--- Backups/Rob4/HOME/Module1.mod ---
MODULE Module1
!PERS tooldata DrillTool:=[TRUE,[[31.792631019,0,229.638935148],[0.945518576,0,0.325568154,0]],[1,[0,0,1],[1,0,0,0],0,0,0]];
PERS tooldata DrillTool:=[TRUE,[[67.056,0,55.372],[0.7071,0,0.7071,0]],[1,[0,0,1],[1,0,0,0],0,0,0]];
PERS wobjdata FakeWing:=[FALSE, TRUE, "",[[-738.2, -596.9, 290],[0.9912, 0, -0.1326, 0]],[[0, 0, 0],[1, 0, 0, 0]]];
!PERS wobjdata FakeWing:=[FALSE, TRUE, "",[[-738.2, -871.22, 290],[1,0,0,0]],[[0, 0, 0],[1, 0, 0, 0]]];
CONST jointtarget jHome:=[[-90,0,28.434410486,3.185484116,-20,-3.571881577],[9E+09,9E+09,9E+09,9E+09,9E+09,9E+09]];
	CONST robtarget Target_10:=[[968.8,4.8,-256.8],[-0.107942386345314,0.559135464335052,0.818413471745805,-0.0769113971910747],[-1,0,0,1],[9E+09,9E+09,9E+09,9E+09,9E+09,9E+09]];
	CONST robtarget Target_20:=[[968.8,9.6,-256.9],[-0.106640376548865,0.55772059756557,0.819364658230691,-0.0788487284813297],[-1,0,0,1],[9E+09,9E+09,9E+09,9E+09,9E+09,9E+09]];
	CONST robtarget Target_30:=[[968.8,14.5,-256.9],[-0.105307817924908,0.556255492926737,0.820340422972373,-0.0808188128484617],[-1,0,0,1],[9E+09,9E+09,9E+09,9E+09,9E+09,9E+09]];
	CONST robtarget Target_40:=[[968.8,19.3,-257],[-0.104018956602322,0.554797112975153,0.821298505042471,-0.0827585990504985],[-1,0,0,1],[9E+09,9E+09,9E+09,9E+09,9E+09,9E+09]];
	CONST robtarget Target_50:=[[968.8,24.1,-257.1],[-0.10270808792262,0.553310583836471,0.822263480299647,-0.0847420524611851],[-1,0,0,1],[9E+09,9E+09,9E+09,9E+09,9E+09,9E+09]];
	CONST robtarget Target_60:=[[968.8,28.9,-257.3],[-0.101414305361901,0.551800115908394,0.823230694611851,-0.0867351958569063],[-1,0,0,1],[9E+09,9E+09,9E+09,9E+09,9E+09,9E+09]];
	CONST robtarget Target_70:=[[968.8,33.7,-257.4],[-0.100146565654331,0.55027415284443,0.824199705211674,-0.0886784530084809],[-1,0,0,1],[9E+09,9E+09,9E+09,9E+09,9E+09,9E+09]];
	CONST robtarget Target_80:=[[968.8,38.5,-257.6],[-0.0988674093110697,0.54871723908215,0.825174424011152,-0.0906741245783206],[-1,0,0,1],[9E+09,9E+09,9E+09,9E+09,9E+09,9E+09]];
	CONST robtarget Target_90:=[[968.8,43.4,-257.8],[-0.0976274781322347,0.547116328064163,0.826167750273506,-0.0926253069476237],[-1,0,0,1],[9E+09,9E+09,9E+09,9E+09,9E+09,9E+09]];
	CONST robtarget Target_100:=[[968.8,48.2,-258.1],[-0.0963734022079838,0.545509328348709,0.827149560398508,-0.0946326833813457],[-1,0,0,1],[9E+09,9E+09,9E+09,9E+09,9E+09,9E+09]];
	CONST robtarget Target_110:=[[968.8,53,-258.3],[-0.0951272887762192,0.543877494214756,0.828135551386225,-0.0966414959890247],[-1,0,0,1],[9E+09,9E+09,9E+09,9E+09,9E+09,9E+09]];
	CONST robtarget Target_120:=[[968.8,57.8,-258.6],[-0.0939178195285495,0.54222699826944,0.82912338791337,-0.0986089911609059],[-1,0,0,1],[9E+09,9E+09,9E+09,9E+09,9E+09,9E+09]];
	CONST robtarget Target_130:=[[968.8,62.6,-258.9],[-0.0926884156537042,0.540544275757953,0.83011823749075,-0.100620352484805],[-1,0,0,1],[9E+09,9E+09,9E+09,9E+09,9E+09,9E+09]];
	CONST robtarget Target_140:=[[968.8,67.4,-259.2],[-0.091496096140411,0.538842149319605,0.831115432114365,-0.102590160390974],[-1,0,0,1],[9E+09,9E+09,9E+09,9E+09,9E+09,9E+09]];
	CONST robtarget Target_150:=[[968.8,72.3,-259.6],[-0.0902970417660465,0.537075607015845,0.832137487086423,-0.104610894185818],[-1,0,0,1],[9E+09,9E+09,9E+09,9E+09,9E+09,9E+09]];
	CONST robtarget Target_160:=[[968.8,77.1,-260],[-0.0891036215361824,0.535310554276655,0.833145780021638,-0.106636130562277],[-1,0,0,1],[9E+09,9E+09,9E+09,9E+09,9E+09,9E+09]];
	CONST robtarget Target_170:=[[968.8,81.9,-260.4],[-0.0879477385246057,0.533524737247738,0.834157223840012,-0.108619869032618],[-1,0,0,1],[9E+09,9E+09,9E+09,9E+09,9E+09,9E+09]];
	CONST robtarget Target_180:=[[968.8,86.7,-260.8],[-0.0867820002749409,0.531701655816364,0.835174793612655,-0.110658473441827],[-1,0,0,1],[9E+09,9E+09,9E+09,9E+09,9E+09,9E+09]];
	CONST robtarget Target_190:=[[968.8,91.5,-261.3],[-0.0856457062027853,0.529858976157848,0.836197037860416,-0.11264453944799],[-1,0,0,1],[9E+09,9E+09,9E+09,9E+09,9E+09,9E+09]];
	CONST robtarget Target_200:=[[968.8,96.3,-261.8],[-0.0845001294653035,0.52797768348931,0.837225467326941,-0.114685704064607],[-1,0,0,1],[9E+09,9E+09,9E+09,9E+09,9E+09,9E+09]];
	CONST robtarget Target_210:=[[968.8,101.2,-262.3],[-0.0833777397174588,0.526031720385176,0.83827881205061,-0.11673651928697],[-1,0,0,1],[9E+09,9E+09,9E+09,9E+09,9E+09,9E+09]];
	CONST robtarget Target_220:=[[968.8,106,-262.8],[-0.0822813203856298,0.524096558354244,0.839317580280092,-0.118737446787462],[-1,0,0,1],[9E+09,9E+09,9E+09,9E+09,9E+09,9E+09]];
	CONST robtarget Target_230:=[[968.8,110.8,-263.4],[-0.0811763419641853,0.522120475519326,0.840362638876055,-0.12079422887729],[-1,0,0,1],[9E+09,9E+09,9E+09,9E+09,9E+09,9E+09]];
	CONST robtarget Target_240:=[[968.8,115.6,-264],[-0.0801102368360122,0.520119946233772,0.841412748073788,-0.122809522687666],[-1,0,0,1],[9E+09,9E+09,9E+09,9E+09,9E+09,9E+09]];
	CONST robtarget Target_250:=[[968.8,120.4,-264.6],[-0.0790283539545263,0.518079466998265,0.842470151681068,-0.124868845884432],[-1,0,0,1],[9E+09,9E+09,9E+09,9E+09,9E+09,9E+09]];
	CONST robtarget Target_260:=[[968.8,125.3,-265.2],[-0.0779715226802002,0.515967795467923,0.843554530052155,-0.126938688032417],[-1,0,0,1],[9E+09,9E+09,9E+09,9E+09,9E+09,9E+09]];
	CONST robtarget Target_270:=[[968.8,130.1,-265.9],[-0.076949075572964,0.513864462728356,0.844623466676326,-0.128970358040245],[-1,0,0,1],[9E+09,9E+09,9E+09,9E+09,9E+09,9E+09]];
	CONST robtarget Target_280:=[[968.8,134.9,-266.6],[-0.0759120858706762,0.511718820666067,0.845699772579321,-0.131046169170174],[-1,0,0,1],[9E+09,9E+09,9E+09,9E+09,9E+09,9E+09]];
	CONST robtarget Target_290:=[[968.8,139.7,-267.3],[-0.0748882393420013,0.509537785767557,0.846782863288632,-0.133123172002685],[-1,0,0,1],[9E+09,9E+09,9E+09,9E+09,9E+09,9E+09]];
	CONST robtarget Target_300:=[[968.8,144.5,-268],[-0.0739120235779645,0.507325477212431,0.847871706099419,-0.135171901436095],[-1,0,0,1],[9E+09,9E+09,9E+09,9E+09,9E+09,9E+09]];
	CONST robtarget Target_310:=[[968.8,149.4,-268.8],[-0.0729217598159667,0.505032843902239,0.848991917508329,-0.137247832518004],[-1,0,0,1],[9E+09,9E+09,9E+09,9E+09,9E+09,9E+09]];
	CONST robtarget Target_320:=[[968.8,154.2,-269.6],[-0.0719805492460282,0.502742088257011,0.850094765604421,-0.139312895014009],[-1,0,0,1],[9E+09,9E+09,9E+09,9E+09,9E+09,9E+09]];
	CONST robtarget Target_330:=[[968.8,159,-270.4],[-0.0710201466278696,0.500407925392313,0.851206058488137,-0.141408249301824],[-1,0,0,1],[9E+09,9E+09,9E+09,9E+09,9E+09,9E+09]];
	CONST robtarget Target_340:=[[968.8,163.8,-271.2],[-0.0701081554829596,0.498039124477821,0.852324167132108,-0.143476099566102],[-1,0,0,1],[9E+09,9E+09,9E+09,9E+09,9E+09,9E+09]];
	CONST robtarget Target_350:=[[968.8,168.6,-272.1],[-0.0691850402824734,0.495621840436952,0.853449773615657,-0.145588136186932],[-1,0,0,1],[9E+09,9E+09,9E+09,9E+09,9E+09,9E+09]];
	CONST robtarget Target_360:=[[968.8,173.4,-273],[-0.0682778424968577,0.493163293359647,0.854583178611091,-0.147701364724926],[-1,0,0,1],[9E+09,9E+09,9E+09,9E+09,9E+09,9E+09]];
	CONST robtarget Target_370:=[[968.8,178.3,-273.9],[-0.0674207080420315,0.490627737512659,0.855749964564331,-0.149769387587943],[-1,0,0,1],[9E+09,9E+09,9E+09,9E+09,9E+09,9E+09]];
	CONST robtarget Target_380:=[[968.8,183.1,-274.9],[-0.0665534629922089,0.488079478410023,0.85689877770681,-0.151899783025914],[-1,0,0,1],[9E+09,9E+09,9E+09,9E+09,9E+09,9E+09]];
	CONST robtarget Target_390:=[[968.8,187.9,-275.8],[-0.0657293478681176,0.485495470345176,0.85805671857293,-0.153988534686852],[-1,0,0,1],[9E+09,9E+09,9E+09,9E+09,9E+09,9E+09]];
	CONST robtarget Target_400:=[[968.8,192.7,-276.8],[-0.0648970915608762,0.482857906815298,0.859222188208384,-0.156121236938751],[-1,0,0,1],[9E+09,9E+09,9E+09,9E+09,9E+09,9E+09]];
	CONST robtarget Target_410:=[[968.8,197.5,-277.9],[-0.0640894833612442,0.480170166912685,0.860394987305689,-0.158270700853872],[-1,0,0,1],[9E+09,9E+09,9E+09,9E+09,9E+09,9E+09]];
	CONST robtarget Target_420:=[[973.5,197.2,-279.1],[-0.0647831891782489,0.476538276592348,0.862417809926292,-0.157955469877521],[-1,0,0,1],[9E+09,9E+09,9E+09,9E+09,9E+09,9E+09]];
	CONST robtarget Target_430:=[[978.2,197,-280.4],[-0.0654513013274054,0.472883025030647,0.864427470973437,-0.157679799653864],[-1,0,0,1],[9E+09,9E+09,9E+09,9E+09,9E+09,9E+09]];
	CONST robtarget Target_440:=[[982.9,196.6,-281.6],[-0.0660933755521842,0.46935615793945,0.866347508185939,-0.157411745979934],[-1,0,0,1],[9E+09,9E+09,9E+09,9E+09,9E+09,9E+09]];
	CONST robtarget Target_450:=[[987.6,196.4,-282.9],[-0.0667443729406992,0.465766124616528,0.86828286007232,-0.157136821735347],[-1,0,0,1],[9E+09,9E+09,9E+09,9E+09,9E+09,9E+09]];
	CONST robtarget Target_460:=[[992.3,196.1,-284.1],[-0.0674028023794809,0.462266046873075,0.870157221438666,-0.156822747450342],[-1,0,0,1],[9E+09,9E+09,9E+09,9E+09,9E+09,9E+09]];
	CONST robtarget Target_470:=[[997.1,195.8,-285.4],[-0.0680417113457267,0.458714001293542,0.87203494948929,-0.156546598186054],[-1,0,0,1],[9E+09,9E+09,9E+09,9E+09,9E+09,9E+09]];
	CONST robtarget Target_480:=[[1001.8,195.5,-286.6],[-0.0686583135132066,0.455272740455241,0.873836494953086,-0.156277150831474],[-1,0,0,1],[9E+09,9E+09,9E+09,9E+09,9E+09,9E+09]];
	CONST robtarget Target_490:=[[1006.5,195.2,-287.9],[-0.0692598520335908,0.451868831293863,0.875604850746204,-0.155992876603775],[-1,0,0,1],[9E+09,9E+09,9E+09,9E+09,9E+09,9E+09]];
	CONST robtarget Target_500:=[[1011.2,194.9,-289.1],[-0.0698599262628231,0.448494319419836,0.877338099476652,-0.155725063356508],[-1,0,0,1],[9E+09,9E+09,9E+09,9E+09,9E+09,9E+09]];
	CONST robtarget Target_510:=[[1015.9,194.6,-290.4],[-0.0704757269732864,0.445161665334504,0.879039624191811,-0.155414293824337],[-1,0,0,1],[9E+09,9E+09,9E+09,9E+09,9E+09,9E+09]];
	CONST robtarget Target_520:=[[1020.6,194.3,-291.6],[-0.0710595030740004,0.441853803362528,0.880706980576819,-0.155148244721643],[-1,0,0,1],[9E+09,9E+09,9E+09,9E+09,9E+09,9E+09]];
	CONST robtarget Target_530:=[[1025.3,194,-292.9],[-0.0716353435846854,0.438579183432016,0.882342262981194,-0.154883208795643],[-1,0,0,1],[9E+09,9E+09,9E+09,9E+09,9E+09,9E+09]];
	CONST robtarget Target_540:=[[1030.1,193.7,-294.1],[-0.0722159183465569,0.435265792974258,0.883981480942423,-0.154613362794727],[-1,0,0,1],[9E+09,9E+09,9E+09,9E+09,9E+09,9E+09]];
	CONST robtarget Target_550:=[[1034.8,193.4,-295.4],[-0.0727991731829624,0.432066562567872,0.885555376103445,-0.15430632439711],[-1,0,0,1],[9E+09,9E+09,9E+09,9E+09,9E+09,9E+09]];
	CONST robtarget Target_560:=[[1039.5,193.1,-296.6],[-0.0733514213142073,0.428891789433335,0.887097329266413,-0.154044572628362],[-1,0,0,1],[9E+09,9E+09,9E+09,9E+09,9E+09,9E+09]];
	CONST robtarget Target_570:=[[1044.2,192.8,-297.9],[-0.0738960968592212,0.425749832850519,0.888609542185254,-0.153784031141213],[-1,0,0,1],[9E+09,9E+09,9E+09,9E+09,9E+09,9E+09]];
	CONST robtarget Target_580:=[[1048.9,192.5,-299.1],[-0.0744560047898698,0.422649013071223,0.890094329524097,-0.153480290753246],[-1,0,0,1],[9E+09,9E+09,9E+09,9E+09,9E+09,9E+09]];
	CONST robtarget Target_590:=[[1053.6,192.3,-300.4],[-0.0749948386695809,0.41951882253895,0.89157392359611,-0.153217722447156],[-1,0,0,1],[9E+09,9E+09,9E+09,9E+09,9E+09,9E+09]];
	CONST robtarget Target_600:=[[1058.4,191.9,-301.6],[-0.0755196426375664,0.416459958972194,0.893006834393729,-0.152959732854318],[-1,0,0,1],[9E+09,9E+09,9E+09,9E+09,9E+09,9E+09]];
	CONST robtarget Target_610:=[[1063.2,191.7,-302.9],[-0.0760553161680778,0.413327332533263,0.894461077902201,-0.152694090198487],[-1,0,0,1],[9E+09,9E+09,9E+09,9E+09,9E+09,9E+09]];
	CONST robtarget Target_620:=[[1063.2,186.7,-301.8],[-0.0766806108289428,0.416479421442643,0.893328220646938,-0.150431597855895],[-1,0,0,1],[9E+09,9E+09,9E+09,9E+09,9E+09,9E+09]];
	CONST robtarget Target_630:=[[1063.2,181.8,-300.8],[-0.0773349992657743,0.419532651685502,0.892221234188017,-0.148165182557526],[-1,0,0,1],[9E+09,9E+09,9E+09,9E+09,9E+09,9E+09]];
	CONST robtarget Target_640:=[[1063.2,176.9,-299.8],[-0.078016434697904,0.422537939615321,0.891114002676915,-0.145914220471464],[-1,0,0,1],[9E+09,9E+09,9E+09,9E+09,9E+09,9E+09]];
	CONST robtarget Target_650:=[[1063.2,172,-298.9],[-0.0787092090169855,0.425503303914037,0.890009339895156,-0.143649481981481],[-1,0,0,1],[9E+09,9E+09,9E+09,9E+09,9E+09,9E+09]];
	CONST robtarget Target_660:=[[1063.2,167.1,-298],[-0.0794359651980819,0.428418799418737,0.888903404145049,-0.141414277344971],[-1,0,0,1],[9E+09,9E+09,9E+09,9E+09,9E+09,9E+09]];
	CONST robtarget Target_670:=[[1063.2,162.2,-297],[-0.080173119410487,0.431295682248896,0.887800214850835,-0.139165670724727],[-1,0,0,1],[9E+09,9E+09,9E+09,9E+09,9E+09,9E+09]];
	CONST robtarget Target_680:=[[1063.2,157.3,-296.2],[-0.0809358269586631,0.434127793589296,0.886697299437008,-0.136931917093582],[-1,0,0,1],[9E+09,9E+09,9E+09,9E+09,9E+09,9E+09]];
	CONST robtarget Target_690:=[[1063.2,152.3,-295.3],[-0.0817086501801631,0.436966661334309,0.885572594947853,-0.134703424030007],[-1,0,0,1],[9E+09,9E+09,9E+09,9E+09,9E+09,9E+09]];
	CONST robtarget Target_700:=[[1063.2,147.4,-294.5],[-0.08250580415254,0.439717260260226,0.884473177381368,-0.13247158866448],[-1,0,0,1],[9E+09,9E+09,9E+09,9E+09,9E+09,9E+09]];
	CONST robtarget Target_710:=[[1063.2,142.5,-293.7],[-0.0833275449806797,0.442425399854024,0.883374314134519,-0.130254009300549],[-1,0,0,1],[9E+09,9E+09,9E+09,9E+09,9E+09,9E+09]];
	CONST robtarget Target_720:=[[1063.2,137.6,-293],[-0.084165466257925,0.445094852551447,0.882277267153493,-0.128037378862409],[-1,0,0,1],[9E+09,9E+09,9E+09,9E+09,9E+09,9E+09]];
	CONST robtarget Target_730:=[[1063.2,132.7,-292.2],[-0.0850191501533236,0.447726204834992,0.881182074536164,-0.125821862676577],[-1,0,0,1],[9E+09,9E+09,9E+09,9E+09,9E+09,9E+09]];
	CONST robtarget Target_740:=[[1063.2,127.8,-291.5],[-0.0859121433611262,0.45032775504269,0.88008875807987,-0.123562917425661],[-1,0,0,1],[9E+09,9E+09,9E+09,9E+09,9E+09,9E+09]];
	CONST robtarget Target_750:=[[1063.2,122.9,-290.8],[-0.086780631442478,0.452874240084196,0.878996243451927,-0.121406954792581],[-1,0,0,1],[9E+09,9E+09,9E+09,9E+09,9E+09,9E+09]];
	CONST robtarget Target_760:=[[1063.2,117.9,-290.2],[-0.0877062031981979,0.455442391239945,0.877883293636171,-0.119166996004373],[-1,0,0,1],[9E+09,9E+09,9E+09,9E+09,9E+09,9E+09]];
	CONST robtarget Target_770:=[[1063.2,113,-289.5],[-0.0886123421515343,0.45791392918028,0.876794047722577,-0.117025143278514],[-1,0,0,1],[9E+09,9E+09,9E+09,9E+09,9E+09,9E+09]];
	CONST robtarget Target_780:=[[1063.2,108.1,-288.9],[-0.0895724613928606,0.460367973564089,0.875707061369707,-0.11478347330409],[-1,0,0,1],[9E+09,9E+09,9E+09,9E+09,9E+09,9E+09]];
	CONST robtarget Target_790:=[[1063.2,103.2,-288.4],[-0.0905306758260853,0.462777522277536,0.874621375658715,-0.112599337697844],[-1,0,0,1],[9E+09,9E+09,9E+09,9E+09,9E+09,9E+09]];
	CONST robtarget Target_800:=[[1063.2,98.3,-287.8],[-0.0914776539191496,0.465145784372994,0.873538533379098,-0.110461164285803],[-1,0,0,1],[9E+09,9E+09,9E+09,9E+09,9E+09,9E+09]];
	CONST robtarget Target_810:=[[1063.2,93.4,-287.3],[-0.0924959019244163,0.467493099310707,0.87245488356131,-0.10824595315336],[-1,0,0,1],[9E+09,9E+09,9E+09,9E+09,9E+09,9E+09]];
	CONST robtarget Target_820:=[[1063.2,88.5,-286.8],[-0.0934775740677943,0.469793072491761,0.871375182242977,-0.106121175814107],[-1,0,0,1],[9E+09,9E+09,9E+09,9E+09,9E+09,9E+09]];
	CONST robtarget Target_830:=[[1063.2,83.5,-286.3],[-0.0945168078179997,0.472113460240636,0.870274451230033,-0.103912623081962],[-1,0,0,1],[9E+09,9E+09,9E+09,9E+09,9E+09,9E+09]];
	CONST robtarget Target_840:=[[1063.2,78.6,-285.9],[-0.0955481155796674,0.47435593029813,0.869197771779048,-0.101745970605763],[-1,0,0,1],[9E+09,9E+09,9E+09,9E+09,9E+09,9E+09]];
	CONST robtarget Target_850:=[[1063.2,73.7,-285.5],[-0.0966006758146477,0.476565156559149,0.868121897640117,-0.0995908219849055],[-1,0,0,1],[9E+09,9E+09,9E+09,9E+09,9E+09,9E+09]];
	CONST robtarget Target_860:=[[1063.2,68.8,-285.1],[-0.0976649286535562,0.47874362573452,0.867047946051864,-0.09743696309361],[-1,0,0,1],[9E+09,9E+09,9E+09,9E+09,9E+09,9E+09]];
	CONST robtarget Target_870:=[[1063.2,63.9,-284.7],[-0.0987405471140935,0.480891783652933,0.865975897316991,-0.0952845319909914],[-1,0,0,1],[9E+09,9E+09,9E+09,9E+09,9E+09,9E+09]];
	CONST robtarget Target_880:=[[1063.2,59,-284.4],[-0.0998272086701067,0.483010067703361,0.864905730830889,-0.0931336656758201],[-1,0,0,1],[9E+09,9E+09,9E+09,9E+09,9E+09,9E+09]];
	CONST robtarget Target_890:=[[1063.2,54.1,-284.1],[-0.100934466374847,0.485097309065803,0.863836217768386,-0.09099353332161],[-1,0,0,1],[9E+09,9E+09,9E+09,9E+09,9E+09,9E+09]];
	CONST robtarget Target_900:=[[1063.2,49.1,-283.8],[-0.102048799399347,0.487190226356418,0.862748992686117,-0.0888588853352571],[-1,0,0,1],[9E+09,9E+09,9E+09,9E+09,9E+09,9E+09]];
	CONST robtarget Target_910:=[[1063.2,44.2,-283.6],[-0.103177151310856,0.4892196127847,0.861683235190265,-0.0867216703379402],[-1,0,0,1],[9E+09,9E+09,9E+09,9E+09,9E+09,9E+09]];
	CONST robtarget Target_920:=[[1063.2,39.3,-283.4],[-0.10432573974925,0.491219543140388,0.860617959114868,-0.0845944969349602],[-1,0,0,1],[9E+09,9E+09,9E+09,9E+09,9E+09,9E+09]];
	CONST robtarget Target_930:=[[1063.2,34.4,-283.2],[-0.105484285502105,0.493191938801291,0.85955435750845,-0.0824686819451414],[-1,0,0,1],[9E+09,9E+09,9E+09,9E+09,9E+09,9E+09]];
	CONST robtarget Target_940:=[[1063.2,29.5,-283],[-0.106652496713291,0.495137184746014,0.858492398121187,-0.0803443563341304],[-1,0,0,1],[9E+09,9E+09,9E+09,9E+09,9E+09,9E+09]];
	CONST robtarget Target_950:=[[1063.2,24.6,-282.8],[-0.107840656413329,0.497054461120178,0.857430708523191,-0.0782293780257217],[-1,0,0,1],[9E+09,9E+09,9E+09,9E+09,9E+09,9E+09]];
	CONST robtarget Target_960:=[[1063.2,19.7,-282.7],[-0.109027458012561,0.498946597101844,0.8563719098455,-0.0761082036798955],[-1,0,0,1],[9E+09,9E+09,9E+09,9E+09,9E+09,9E+09]];
	CONST robtarget Target_970:=[[1063.2,14.7,-282.6],[-0.110231181610952,0.500842889389237,0.855294950614735,-0.0740002310930915],[-1,0,0,1],[9E+09,9E+09,9E+09,9E+09,9E+09,9E+09]];
	CONST robtarget Target_980:=[[1063.2,9.8,-282.6],[-0.111457441458863,0.502680910869204,0.854236489571451,-0.0718968738944611],[-1,0,0,1],[9E+09,9E+09,9E+09,9E+09,9E+09,9E+09]];
	CONST robtarget Target_990:=[[1063.2,4.9,-282.5],[-0.112681393063629,0.504494799312451,0.853180840830537,-0.0697879213304613],[-1,0,0,1],[9E+09,9E+09,9E+09,9E+09,9E+09,9E+09]];
	CONST robtarget Target_1000:=[[1067.8,0,-283.8],[-0.11412479964084,0.503756290219997,0.853621201330236,-0.0673496459548792],[-1,0,0,1],[9E+09,9E+09,9E+09,9E+09,9E+09,9E+09]];
	CONST robtarget Target_1010:=[[1072.5,0,-285.1],[-0.114326804980448,0.501187162072787,0.855132144098277,-0.067006166628692],[-1,0,0,1],[9E+09,9E+09,9E+09,9E+09,9E+09,9E+09]];
	CONST robtarget Target_1020:=[[1077.2,0,-286.3],[-0.114526435240778,0.498630738220601,0.856625321945522,-0.0666643858019352],[-1,0,0,1],[9E+09,9E+09,9E+09,9E+09,9E+09,9E+09]];
	CONST robtarget Target_1030:=[[1081.9,0,-287.6],[-0.114723708623628,0.496087139984326,0.858100871016259,-0.0663243196945924],[-1,0,0,1],[9E+09,9E+09,9E+09,9E+09,9E+09,9E+09]];
	CONST robtarget Target_1040:=[[1086.7,0,-288.9],[-0.114922765954398,0.493502779892004,0.859589763512546,-0.0659788039350536],[-1,0,0,1],[9E+09,9E+09,9E+09,9E+09,9E+09,9E+09]];
	CONST robtarget Target_1050:=[[1091.4,0,-290.2],[-0.11511533237106,0.49098545007799,0.861030105808388,-0.0656422497817516],[-1,0,0,1],[9E+09,9E+09,9E+09,9E+09,9E+09,9E+09]];
	CONST robtarget Target_1060:=[[1096.1,0,-291.5],[-0.115305598862751,0.488481273888714,0.862453245316376,-0.0653074542009705],[-1,0,0,1],[9E+09,9E+09,9E+09,9E+09,9E+09,9E+09]];
	CONST robtarget Target_1070:=[[1100.8,0,-292.8],[-0.115493584857007,0.485990347485264,0.863859327348986,-0.064974430048957],[-1,0,0,1],[9E+09,9E+09,9E+09,9E+09,9E+09,9E+09]];
	CONST robtarget Target_1080:=[[1105.5,0,-294],[-0.115679310033985,0.483512761039106,0.865248499108222,-0.064643189381176],[-1,0,0,1],[9E+09,9E+09,9E+09,9E+09,9E+09,9E+09]];
	CONST robtarget Target_1090:=[[1110.2,0,-295.3],[-0.115862794306681,0.481048598843016,0.866620909537649,-0.0643137434671416],[-1,0,0,1],[9E+09,9E+09,9E+09,9E+09,9E+09,9E+09]];
	CONST robtarget Target_1100:=[[1115,0,-296.6],[-0.116047890492229,0.478545944980402,0.868005376619007,-0.0639791514136686],[-1,0,0,1],[9E+09,9E+09,9E+09,9E+09,9E+09,9E+09]];
	CONST robtarget Target_1110:=[[1119.7,0,-297.9],[-0.116226906934761,0.476109150808135,0.869344368943313,-0.0636533644647941],[-1,0,0,1],[9E+09,9E+09,9E+09,9E+09,9E+09,9E+09]];
	CONST robtarget Target_1120:=[[1124.4,0,-299.2],[-0.116403743856853,0.473686001001012,0.870667059071583,-0.063329401697929],[-1,0,0,1],[9E+09,9E+09,9E+09,9E+09,9E+09,9E+09]];
	CONST robtarget Target_1130:=[[1129.1,0,-300.5],[-0.116578421918569,0.471276557365558,0.871973601535252,-0.0630072713762903],[-1,0,0,1],[9E+09,9E+09,9E+09,9E+09,9E+09,9E+09]];
	CONST robtarget Target_1140:=[[1133.8,0,-301.7],[-0.116750961921334,0.468880876409721,0.873264151923084,-0.0626869810547025],[-1,0,0,1],[9E+09,9E+09,9E+09,9E+09,9E+09,9E+09]];
	CONST robtarget Target_1150:=[[1138.6,0,-303],[-0.11692498796171,0.46644848187319,0.874565817451658,-0.0623617823146801],[-1,0,0,1],[9E+09,9E+09,9E+09,9E+09,9E+09,9E+09]];
	CONST robtarget Target_1160:=[[1143.3,0,-304.3],[-0.117093270365041,0.464080770565376,0.87582452220073,-0.0620452313923381],[-1,0,0,1],[9E+09,9E+09,9E+09,9E+09,9E+09,9E+09]];
	CONST robtarget Target_1170:=[[1148,0,-305.6],[-0.11725947824855,0.461726961684459,0.877067710128658,-0.0617305391535456],[-1,0,0,1],[9E+09,9E+09,9E+09,9E+09,9E+09,9E+09]];
	CONST robtarget Target_1180:=[[1152.7,0,-306.9],[-0.11742363281949,0.459387091633213,0.878295539859715,-0.0614177104651672],[-1,0,0,1],[9E+09,9E+09,9E+09,9E+09,9E+09,9E+09]];
	CONST robtarget Target_1190:=[[1157.5,4.9,-308.2],[-0.116456698651549,0.454978592783004,0.880583191851778,-0.0632894910432632],[-1,0,0,1],[9E+09,9E+09,9E+09,9E+09,9E+09,9E+09]];
	CONST robtarget Target_1200:=[[1157.5,9.8,-308.2],[-0.115321553262797,0.452913443093735,0.881632492180146,-0.0655324434937342],[-1,0,0,1],[9E+09,9E+09,9E+09,9E+09,9E+09,9E+09]];
	CONST robtarget Target_1210:=[[1157.5,14.7,-308.3],[-0.114208395342144,0.450830345502874,0.88267875116301,-0.0677249160386389],[-1,0,0,1],[9E+09,9E+09,9E+09,9E+09,9E+09,9E+09]];
	CONST robtarget Target_1220:=[[1157.5,19.6,-308.4],[-0.113116403345818,0.448720948594571,0.883722022425974,-0.0699255079769918],[-1,0,0,1],[9E+09,9E+09,9E+09,9E+09,9E+09,9E+09]];
	CONST robtarget Target_1230:=[[1157.5,24.4,-308.5],[-0.112042503144085,0.44662162946331,0.884743749945618,-0.0721394102894673],[-1,0,0,1],[9E+09,9E+09,9E+09,9E+09,9E+09,9E+09]];
	CONST robtarget Target_1240:=[[1157.5,29.3,-308.7],[-0.110947538224501,0.444454570827599,0.885786132357125,-0.0743888832836221],[-1,0,0,1],[9E+09,9E+09,9E+09,9E+09,9E+09,9E+09]];
	CONST robtarget Target_1250:=[[1157.5,34.2,-308.8],[-0.109897288481995,0.442266525786448,0.886823054715504,-0.0766014084606349],[-1,0,0,1],[9E+09,9E+09,9E+09,9E+09,9E+09,9E+09]];
	CONST robtarget Target_1260:=[[1157.5,39.1,-309.1],[-0.10886840289795,0.4400505689674,0.887857005220818,-0.0788232572419922],[-1,0,0,1],[9E+09,9E+09,9E+09,9E+09,9E+09,9E+09]];
	CONST robtarget Target_1270:=[[1157.5,44,-309.3],[-0.107839723601408,0.437809013192539,0.888890636361769,-0.0810388707307653],[-1,0,0,1],[9E+09,9E+09,9E+09,9E+09,9E+09,9E+09]];
	CONST robtarget Target_1280:=[[1157.5,48.9,-309.5],[-0.106809880606017,0.435532061690535,0.889922999304026,-0.0833098310780098],[-1,0,0,1],[9E+09,9E+09,9E+09,9E+09,9E+09,9E+09]];
	CONST robtarget Target_1290:=[[1157.5,53.8,-309.8],[-0.105814334622865,0.433234255109494,0.890951696495378,-0.0855364325889902],[-1,0,0,1],[9E+09,9E+09,9E+09,9E+09,9E+09,9E+09]];
	CONST robtarget Target_1300:=[[1157.5,58.7,-310.1],[-0.104830406221372,0.430908588307866,0.891978581406433,-0.0877643707101632],[-1,0,0,1],[9E+09,9E+09,9E+09,9E+09,9E+09,9E+09]];
	CONST robtarget Target_1310:=[[1157.5,63.6,-310.5],[-0.103868543102495,0.428553079264927,0.893002320186698,-0.090002445230613],[-1,0,0,1],[9E+09,9E+09,9E+09,9E+09,9E+09,9E+09]];
	CONST robtarget Target_1320:=[[1157.5,68.5,-310.8],[-0.102896186994666,0.42616193510684,0.894025342835322,-0.0922879522805532],[-1,0,0,1],[9E+09,9E+09,9E+09,9E+09,9E+09,9E+09]];
	CONST robtarget Target_1330:=[[1157.5,73.3,-311.2],[-0.101954320538193,0.423790577515119,0.89502528752291,-0.0945335793648495],[-1,0,0,1],[9E+09,9E+09,9E+09,9E+09,9E+09,9E+09]];
	CONST robtarget Target_1340:=[[1157.5,78.2,-311.6],[-0.101039180167052,0.421346926627475,0.896041552749548,-0.0967852635421828],[-1,0,0,1],[9E+09,9E+09,9E+09,9E+09,9E+09,9E+09]];
	CONST robtarget Target_1350:=[[1157.5,83.1,-312.1],[-0.100136755641848,0.418873626645508,0.897055691069865,-0.0990383874542113],[-1,0,0,1],[9E+09,9E+09,9E+09,9E+09,9E+09,9E+09]];
	CONST robtarget Target_1360:=[[1157.5,88,-312.6],[-0.0992252665873052,0.416363081924884,0.898068247921142,-0.101338800844204],[-1,0,0,1],[9E+09,9E+09,9E+09,9E+09,9E+09,9E+09]];
	CONST robtarget Target_1370:=[[1157.5,92.9,-313.1],[-0.0983493052491232,0.413829493044003,0.899077740529287,-0.103594311275819],[-1,0,0,1],[9E+09,9E+09,9E+09,9E+09,9E+09,9E+09]];
	CONST robtarget Target_1380:=[[1157.5,97.8,-313.6],[-0.0974965183603951,0.411263091531744,0.900083594760464,-0.10586132860698],[-1,0,0,1],[9E+09,9E+09,9E+09,9E+09,9E+09,9E+09]];
	CONST robtarget Target_1390:=[[1157.5,102.7,-314.2],[-0.0966575256864694,0.408665629753412,0.901086967457954,-0.108129565169957],[-1,0,0,1],[9E+09,9E+09,9E+09,9E+09,9E+09,9E+09]];
	CONST robtarget Target_1400:=[[1157.5,107.6,-314.7],[-0.0958203709921909,0.406026876380138,0.902086535754033,-0.11045593769099],[-1,0,0,1],[9E+09,9E+09,9E+09,9E+09,9E+09,9E+09]];
	CONST robtarget Target_1410:=[[1157.5,112.4,-315.4],[-0.0950042127207623,0.403412314824983,0.903063888470925,-0.112731172053829],[-1,0,0,1],[9E+09,9E+09,9E+09,9E+09,9E+09,9E+09]];
	CONST robtarget Target_1420:=[[1157.5,117.3,-316],[-0.0942176050684812,0.400717638074019,0.904057659766507,-0.115013761129028],[-1,0,0,1],[9E+09,9E+09,9E+09,9E+09,9E+09,9E+09]];
	CONST robtarget Target_1430:=[[1157.5,122.2,-316.7],[-0.0934459398585867,0.397990450533941,0.90504850520611,-0.117297318093474],[-1,0,0,1],[9E+09,9E+09,9E+09,9E+09,9E+09,9E+09]];
	CONST robtarget Target_1440:=[[1157.5,127.1,-317.4],[-0.09267744685106,0.395219958040731,0.906034447792381,-0.119639688335463],[-1,0,0,1],[9E+09,9E+09,9E+09,9E+09,9E+09,9E+09]];
	CONST robtarget Target_1450:=[[1157.5,132,-318.1],[-0.091945722049869,0.392423813800334,0.907017578768495,-0.121937059026639],[-1,0,0,1],[9E+09,9E+09,9E+09,9E+09,9E+09,9E+09]];
	CONST robtarget Target_1460:=[[1157.5,136.9,-318.8],[-0.0912298198832608,0.389593997110689,0.907997372118494,-0.124235299352858],[-1,0,0,1],[9E+09,9E+09,9E+09,9E+09,9E+09,9E+09]];
	CONST robtarget Target_1470:=[[1157.5,141.8,-319.6],[-0.090538948270863,0.386727190520538,0.908972312148108,-0.126546887382584],[-1,0,0,1],[9E+09,9E+09,9E+09,9E+09,9E+09,9E+09]];
	CONST robtarget Target_1480:=[[1157.5,146.7,-320.4],[-0.0898350121694737,0.383820989667297,0.909943857926704,-0.128892567282967],[-1,0,0,1],[9E+09,9E+09,9E+09,9E+09,9E+09,9E+09]];
	CONST robtarget Target_1490:=[[1157.5,151.6,-321.2],[-0.0891774776768113,0.380884851594658,0.910911188916038,-0.131205614241488],[-1,0,0,1],[9E+09,9E+09,9E+09,9E+09,9E+09,9E+09]];
	CONST robtarget Target_1500:=[[1157.5,156.5,-322.1],[-0.0885457305098963,0.377910274200135,0.911873087948939,-0.133532579309003],[-1,0,0,1],[9E+09,9E+09,9E+09,9E+09,9E+09,9E+09]];
	CONST robtarget Target_1510:=[[1157.5,161.3,-323],[-0.087923551535875,0.374952346833089,0.912809279452066,-0.135865396756779],[-1,0,0,1],[9E+09,9E+09,9E+09,9E+09,9E+09,9E+09]];
	CONST robtarget Target_1520:=[[1157.5,166.2,-323.9],[-0.0873065476042629,0.371898546178329,0.913760797007033,-0.138239805949448],[-1,0,0,1],[9E+09,9E+09,9E+09,9E+09,9E+09,9E+09]];
	CONST robtarget Target_1530:=[[1157.5,171.1,-324.9],[-0.0867279055318608,0.368816467199481,0.914709329423617,-0.140568583225226],[-1,0,0,1],[9E+09,9E+09,9E+09,9E+09,9E+09,9E+09]];
	CONST robtarget Target_1540:=[[1157.5,176,-325.8],[-0.0861677390911265,0.365697677609429,0.915653113093589,-0.142897536063477],[-1,0,0,1],[9E+09,9E+09,9E+09,9E+09,9E+09,9E+09]];
	CONST robtarget Target_1550:=[[1157.5,180.9,-326.9],[-0.085634841189232,0.362538132200784,0.916590329863401,-0.145240985523245],[-1,0,0,1],[9E+09,9E+09,9E+09,9E+09,9E+09,9E+09]];
	CONST robtarget Target_1560:=[[1157.5,185.8,-327.9],[-0.0851099118523378,0.359328899108832,0.917518335176831,-0.147645351379778],[-1,0,0,1],[9E+09,9E+09,9E+09,9E+09,9E+09,9E+09]];
	CONST robtarget Target_1570:=[[1162.1,185.5,-329.1],[-0.0855047583298773,0.357001363171177,0.91843204244788,-0.147382313735012],[-1,0,0,1],[9E+09,9E+09,9E+09,9E+09,9E+09,9E+09]];
	CONST robtarget Target_1580:=[[1166.9,185.2,-330.4],[-0.0858922351502221,0.354583671052544,0.919368158097704,-0.147156834839008],[-1,0,0,1],[9E+09,9E+09,9E+09,9E+09,9E+09,9E+09]];
	CONST robtarget Target_1590:=[[1171.6,184.9,-331.6],[-0.0862659090477359,0.352246251074069,0.920266248704867,-0.146938092525744],[-1,0,0,1],[9E+09,9E+09,9E+09,9E+09,9E+09,9E+09]];
	CONST robtarget Target_1600:=[[1176.3,184.6,-332.9],[-0.0866260223795731,0.349938460600053,0.921149417827701,-0.146706360036797],[-1,0,0,1],[9E+09,9E+09,9E+09,9E+09,9E+09,9E+09]];
	CONST robtarget Target_1610:=[[1181,184.3,-334.1],[-0.0870086276767732,0.34766071109707,0.922017047874772,-0.146444843192153],[-1,0,0,1],[9E+09,9E+09,9E+09,9E+09,9E+09,9E+09]];
	CONST robtarget Target_1620:=[[1185.7,184,-335.4],[-0.0873672830921968,0.34539992640377,0.922866348640203,-0.146231156847156],[-1,0,0,1],[9E+09,9E+09,9E+09,9E+09,9E+09,9E+09]];
	CONST robtarget Target_1630:=[[1190.4,183.7,-336.6],[-0.0877211398640291,0.343164103234253,0.923700062175846,-0.146019159731608],[-1,0,0,1],[9E+09,9E+09,9E+09,9E+09,9E+09,9E+09]];
	CONST robtarget Target_1640:=[[1195.1,183.4,-337.9],[-0.0880702742574934,0.340952949211184,0.924518519574609,-0.145808848085359],[-1,0,0,1],[9E+09,9E+09,9E+09,9E+09,9E+09,9E+09]];
	CONST robtarget Target_1650:=[[1199.9,183.2,-339.1],[-0.0884498527767347,0.338669042814087,0.925363124454556,-0.145543776517121],[-1,0,0,1],[9E+09,9E+09,9E+09,9E+09,9E+09,9E+09]];
	CONST robtarget Target_1660:=[[1204.6,182.9,-340.4],[-0.0887895322356481,0.336506913219425,0.926151569677687,-0.145336802993827],[-1,0,0,1],[9E+09,9E+09,9E+09,9E+09,9E+09,9E+09]];
	CONST robtarget Target_1670:=[[1209.3,182.6,-341.6],[-0.0891247139754168,0.334368581224392,0.926925716846229,-0.145131501397497],[-1,0,0,1],[9E+09,9E+09,9E+09,9E+09,9E+09,9E+09]];
	CONST robtarget Target_1680:=[[1214,182.3,-342.9],[-0.0894554700034203,0.332253759117089,0.927685869361753,-0.144927865593746],[-1,0,0,1],[9E+09,9E+09,9E+09,9E+09,9E+09,9E+09]];
	CONST robtarget Target_1690:=[[1218.7,182,-344.1],[-0.0897999545630442,0.330170396324356,0.928434900091322,-0.144679348367038],[-1,0,0,1],[9E+09,9E+09,9E+09,9E+09,9E+09,9E+09]];
	CONST robtarget Target_1700:=[[1223.4,181.7,-345.4],[-0.090121967225503,0.328101731588239,0.92916796546446,-0.144478983616444],[-1,0,0,1],[9E+09,9E+09,9E+09,9E+09,9E+09,9E+09]];
	CONST robtarget Target_1710:=[[1228.2,181.4,-346.6],[-0.0904470279388317,0.326008912409632,0.929904319457681,-0.144275711124456],[-1,0,0,1],[9E+09,9E+09,9E+09,9E+09,9E+09,9E+09]];
	CONST robtarget Target_1720:=[[1232.9,181.1,-347.9],[-0.0907783627727378,0.323993976593036,0.930613762368532,-0.144032000867925],[-1,0,0,1],[9E+09,9E+09,9E+09,9E+09,9E+09,9E+09]];
	CONST robtarget Target_1730:=[[1237.6,180.8,-349.1],[-0.091087744358842,0.321992909345137,0.931308025257883,-0.143836543511497],[-1,0,0,1],[9E+09,9E+09,9E+09,9E+09,9E+09,9E+09]];
	CONST robtarget Target_1740:=[[1242.3,180.5,-350.4],[-0.0913931135312284,0.320013657728264,0.931989984090849,-0.143642706813763],[-1,0,0,1],[9E+09,9E+09,9E+09,9E+09,9E+09,9E+09]];
	CONST robtarget Target_1750:=[[1247,180.2,-351.6],[-0.0916945348607215,0.318055947587207,0.932659898238735,-0.14345048169453],[-1,0,0,1],[9E+09,9E+09,9E+09,9E+09,9E+09,9E+09]];
	CONST robtarget Target_1760:=[[1251.8,179.9,-352.9],[-0.0920162744058036,0.316083234550579,0.93333577734982,-0.143208661746861],[-1,0,0,1],[9E+09,9E+09,9E+09,9E+09,9E+09,9E+09]];
	CONST robtarget Target_1770:=[[1251.8,174.9,-351.8],[-0.0924700063181994,0.319309051540198,0.932576424639331,-0.14068489521954],[-1,0,0,1],[9E+09,9E+09,9E+09,9E+09,9E+09,9E+09]];
	CONST robtarget Target_1780:=[[1251.8,169.9,-350.8],[-0.0929425081399444,0.32250343302878,0.931807201758761,-0.138161371648576],[-1,0,0,1],[9E+09,9E+09,9E+09,9E+09,9E+09,9E+09]];
	CONST robtarget Target_1790:=[[1251.8,164.9,-349.8],[-0.093442636575496,0.325663071896759,0.931026631224141,-0.13565194146791],[-1,0,0,1],[9E+09,9E+09,9E+09,9E+09,9E+09,9E+09]];
	CONST robtarget Target_1800:=[[1251.8,159.9,-348.9],[-0.0939609701945678,0.328791703294963,0.930236719612129,-0.13314277077543],[-1,0,0,1],[9E+09,9E+09,9E+09,9E+09,9E+09,9E+09]];
	CONST robtarget Target_1810:=[[1251.8,154.9,-347.9],[-0.0945064640355247,0.331886219394539,0.929436051575064,-0.130647203047202],[-1,0,0,1],[9E+09,9E+09,9E+09,9E+09,9E+09,9E+09]];
	CONST robtarget Target_1820:=[[1251.8,149.9,-347],[-0.0950696189951441,0.334950171594067,0.928626534887739,-0.128151897354718],[-1,0,0,1],[9E+09,9E+09,9E+09,9E+09,9E+09,9E+09]];
	CONST robtarget Target_1830:=[[1251.8,144.9,-346.2],[-0.0956501185125098,0.337983693851527,0.927808369679983,-0.125657099563821],[-1,0,0,1],[9E+09,9E+09,9E+09,9E+09,9E+09,9E+09]];
	CONST robtarget Target_1840:=[[1251.8,139.9,-345.3],[-0.0962570810498641,0.34098396955735,0.926980220358796,-0.123175394930279],[-1,0,0,1],[9E+09,9E+09,9E+09,9E+09,9E+09,9E+09]];
	CONST robtarget Target_1850:=[[1251.8,135,-344.5],[-0.0968873632454575,0.343904438079092,0.92616237743372,-0.120688967760798],[-1,0,0,1],[9E+09,9E+09,9E+09,9E+09,9E+09,9E+09]];
	CONST robtarget Target_1860:=[[1251.8,129.9,-343.7],[-0.0975211682067817,0.346894770108699,0.925299498644537,-0.118213696461056],[-1,0,0,1],[9E+09,9E+09,9E+09,9E+09,9E+09,9E+09]];
	CONST robtarget Target_1870:=[[1251.8,124.9,-343],[-0.0981776698665501,0.349805589833328,0.92444729188497,-0.115734173809971],[-1,0,0,1],[9E+09,9E+09,9E+09,9E+09,9E+09,9E+09]];
	CONST robtarget Target_1880:=[[1251.8,119.9,-342.3],[-0.0988787294896709,0.35269196810532,0.923586796329145,-0.113220148979633],[-1,0,0,1],[9E+09,9E+09,9E+09,9E+09,9E+09,9E+09]];
	CONST robtarget Target_1890:=[[1251.8,114.9,-341.6],[-0.099586379320185,0.355538933266474,0.922716476741266,-0.110765172937249],[-1,0,0,1],[9E+09,9E+09,9E+09,9E+09,9E+09,9E+09]];
	CONST robtarget Target_1900:=[[1251.8,110,-340.9],[-0.100305303113894,0.358312203741803,0.921858683650493,-0.108294866891757],[-1,0,0,1],[9E+09,9E+09,9E+09,9E+09,9E+09,9E+09]];
	CONST robtarget Target_1910:=[[1251.8,105,-340.3],[-0.101043481429939,0.361102035827114,0.920973980379984,-0.105841683873036],[-1,0,0,1],[9E+09,9E+09,9E+09,9E+09,9E+09,9E+09]];
	CONST robtarget Target_1920:=[[1251.8,99.9,-339.7],[-0.101791401265309,0.363909591209621,0.920064048057718,-0.103394717107482],[-1,0,0,1],[9E+09,9E+09,9E+09,9E+09,9E+09,9E+09]];
	CONST robtarget Target_1930:=[[1251.8,94.9,-339.1],[-0.102569367780589,0.366639855644028,0.919164307545986,-0.10095403300475],[-1,0,0,1],[9E+09,9E+09,9E+09,9E+09,9E+09,9E+09]];
	CONST robtarget Target_1940:=[[1251.8,90,-338.6],[-0.103366683650324,0.369296805579684,0.91827616664258,-0.0985092882726507],[-1,0,0,1],[9E+09,9E+09,9E+09,9E+09,9E+09,9E+09]];
	CONST robtarget Target_1950:=[[1251.8,85,-338.1],[-0.104173173517156,0.371971651231437,0.917363299170589,-0.0960709005598221],[-1,0,0,1],[9E+09,9E+09,9E+09,9E+09,9E+09,9E+09]];
	CONST robtarget Target_1960:=[[1251.8,80,-337.6],[-0.105003845112194,0.374616877120583,0.91644275072051,-0.0936433261898658],[-1,0,0,1],[9E+09,9E+09,9E+09,9E+09,9E+09,9E+09]];
	CONST robtarget Target_1970:=[[1251.8,75,-337.1],[-0.105848296774295,0.377234732453949,0.91551601122939,-0.0912169276121816],[-1,0,0,1],[9E+09,9E+09,9E+09,9E+09,9E+09,9E+09]];
	CONST robtarget Target_1980:=[[1251.8,70,-336.7],[-0.106706240839152,0.379825387564897,0.914583210758717,-0.0887919125001225],[-1,0,0,1],[9E+09,9E+09,9E+09,9E+09,9E+09,9E+09]];
	CONST robtarget Target_1990:=[[1251.8,65,-336.3],[-0.10758792134765,0.382387338002196,0.913643125034888,-0.086377097613721],[-1,0,0,1],[9E+09,9E+09,9E+09,9E+09,9E+09,9E+09]];
	CONST robtarget Target_2000:=[[1251.8,60,-336],[-0.108482698248023,0.384922590330042,0.912697222791255,-0.0839635822459261],[-1,0,0,1],[9E+09,9E+09,9E+09,9E+09,9E+09,9E+09]];
	CONST robtarget Target_2010:=[[1251.8,55,-335.6],[-0.109390290202297,0.38743131692568,0.911745622822499,-0.0815515685851842],[-1,0,0,1],[9E+09,9E+09,9E+09,9E+09,9E+09,9E+09]];
	CONST robtarget Target_2020:=[[1251.8,50,-335.3],[-0.110310416782409,0.389913691291365,0.910788442329569,-0.0791412573296013],[-1,0,0,1],[9E+09,9E+09,9E+09,9E+09,9E+09,9E+09]];
	CONST robtarget Target_2030:=[[1251.8,45,-335],[-0.111253696234398,0.392368519801423,0.909824411361592,-0.0767404732429802],[-1,0,0,1],[9E+09,9E+09,9E+09,9E+09,9E+09,9E+09]];
	CONST robtarget Target_2040:=[[1251.8,40,-334.8],[-0.112240868163906,0.394802969552821,0.90885194146769,-0.0743017579637067],[-1,0,0,1],[9E+09,9E+09,9E+09,9E+09,9E+09,9E+09]];
	CONST robtarget Target_2050:=[[1251.8,35,-334.6],[-0.113208396368411,0.397206277971363,0.907877096868025,-0.0719041634004291],[-1,0,0,1],[9E+09,9E+09,9E+09,9E+09,9E+09,9E+09]];
	CONST robtarget Target_2060:=[[1251.8,30,-334.4],[-0.114177826229758,0.399576296492031,0.906897618349547,-0.0695623253714255],[-1,0,0,1],[9E+09,9E+09,9E+09,9E+09,9E+09,9E+09]];
	CONST robtarget Target_2070:=[[1251.8,25,-334.2],[-0.115200628095068,0.401934408304075,0.905909111119453,-0.0671284522279307],[-1,0,0,1],[9E+09,9E+09,9E+09,9E+09,9E+09,9E+09]];
	CONST robtarget Target_2080:=[[1251.8,20,-334.1],[-0.116225198631262,0.404259867017925,0.904916092191274,-0.0647497429728289],[-1,0,0,1],[9E+09,9E+09,9E+09,9E+09,9E+09,9E+09]];
	CONST robtarget Target_2090:=[[1251.8,15,-334],[-0.117260990851089,0.406560628716403,0.903918121285456,-0.0623726319319307],[-1,0,0,1],[9E+09,9E+09,9E+09,9E+09,9E+09,9E+09]];
	CONST robtarget Target_2100:=[[1251.8,10,-333.9],[-0.118307741993707,0.408836865218115,0.902915288829416,-0.0599973084485274],[-1,0,0,1],[9E+09,9E+09,9E+09,9E+09,9E+09,9E+09]];
	CONST robtarget Target_2110:=[[1251.8,5,-333.9],[-0.119365190355739,0.411088748585182,0.901907684450129,-0.0576239607091761],[-1,0,0,1],[9E+09,9E+09,9E+09,9E+09,9E+09,9E+09]];
	CONST robtarget Target_2120:=[[1256.5,0,-335.1],[-0.120569119039261,0.411284617526314,0.901822886537553,-0.0549866550847202],[-1,0,0,1],[9E+09,9E+09,9E+09,9E+09,9E+09,9E+09]];
	CONST robtarget Target_2130:=[[1261.2,0,-336.4],[-0.1206917614149,0.409267218665977,0.902740216796674,-0.0547169391493933],[-1,0,0,1],[9E+09,9E+09,9E+09,9E+09,9E+09,9E+09]];
	CONST robtarget Target_2140:=[[1265.9,0,-337.7],[-0.120812853870801,0.407263483441308,0.903645954094822,-0.0544490499724465],[-1,0,0,1],[9E+09,9E+09,9E+09,9E+09,9E+09,9E+09]];
	CONST robtarget Target_2150:=[[1270.6,0,-339],[-0.120932416047713,0.405273364358332,0.904540245339238,-0.0541829812041777],[-1,0,0,1],[9E+09,9E+09,9E+09,9E+09,9E+09,9E+09]];
	CONST robtarget Target_2160:=[[1275.3,0,-340.3],[-0.121050467432942,0.403296811893955,0.905423236289451,-0.0539187262236019],[-1,0,0,1],[9E+09,9E+09,9E+09,9E+09,9E+09,9E+09]];
	CONST robtarget Target_2170:=[[1280.1,0,-341.5],[-0.121169491291304,0.401292154280101,0.906313501063471,-0.053650713727927],[-1,0,0,1],[9E+09,9E+09,9E+09,9E+09,9E+09,9E+09]];
	CONST robtarget Target_2180:=[[1284.8,0,-342.8],[-0.12128454780413,0.399342864620878,0.907174091215728,-0.0533901036453117],[-1,0,0,1],[9E+09,9E+09,9E+09,9E+09,9E+09,9E+09]];
	CONST robtarget Target_2190:=[[1289.5,0,-344.1],[-0.121398151432152,0.397406980488293,0.908023814200854,-0.0531312858132162],[-1,0,0,1],[9E+09,9E+09,9E+09,9E+09,9E+09,9E+09]];
	CONST robtarget Target_2200:=[[1294.2,0,-345.4],[-0.121510321009731,0.395484445041252,0.908862810894529,-0.0528742526322758],[-1,0,0,1],[9E+09,9E+09,9E+09,9E+09,9E+09,9E+09]];
	CONST robtarget Target_2210:=[[1298.9,0,-346.7],[-0.121621075201248,0.393575199818587,0.909691220901054,-0.052618996286531],[-1,0,0,1],[9E+09,9E+09,9E+09,9E+09,9E+09,9E+09]];
	CONST robtarget Target_2220:=[[1303.6,0,-348],[-0.121730432498577,0.391679184814837,0.910509182534408,-0.0523655087535576],[-1,0,0,1],[9E+09,9E+09,9E+09,9E+09,9E+09,9E+09]];
	CONST robtarget Target_2230:=[[1308.4,0,-349.3],[-0.121840693793714,0.389756420611296,0.911333905815514,-0.0521084449890404],[-1,0,0,1],[9E+09,9E+09,9E+09,9E+09,9E+09,9E+09]];
	CONST robtarget Target_2240:=[[1313.1,0,-350.5],[-0.121947283327268,0.38788695837475,0.912131165359169,-0.0518585074255761],[-1,0,0,1],[9E+09,9E+09,9E+09,9E+09,9E+09,9E+09]];
	CONST robtarget Target_2250:=[[1317.8,0,-351.8],[-0.122052530765466,0.386030536424691,0.912918386409407,-0.0516103132818866],[-1,0,0,1],[9E+09,9E+09,9E+09,9E+09,9E+09,9E+09]];
	CONST robtarget Target_2260:=[[1322.5,0,-353.1],[-0.122156453885429,0.384187089272802,0.913695701934064,-0.051363853802518],[-1,0,0,1],[9E+09,9E+09,9E+09,9E+09,9E+09,9E+09]];
	CONST robtarget Target_2270:=[[1327.2,0,-354.4],[-0.122259070282356,0.382356550238858,0.914463243540237,-0.0511191200726645],[-1,0,0,1],[9E+09,9E+09,9E+09,9E+09,9E+09,9E+09]];
	CONST robtarget Target_2280:=[[1331.9,0,-355.7],[-0.122360397368242,0.380538851515419,0.915221141464737,-0.0508761030268172],[-1,0,0,1],[9E+09,9E+09,9E+09,9E+09,9E+09,9E+09]];
	CONST robtarget Target_2290:=[[1336.6,0,-357],[-0.122460452370791,0.378733924230739,0.915969524565897,-0.0506347934571751],[-1,0,0,1],[9E+09,9E+09,9E+09,9E+09,9E+09,9E+09]];
	CONST robtarget Target_2300:=[[1341.4,0,-358.2],[-0.122561340947479,0.376903703528983,0.916724142565705,-0.050390102286711],[-1,0,0,1],[9E+09,9E+09,9E+09,9E+09,9E+09,9E+09]];
	CONST robtarget Target_2310:=[[1346.2,5,-359.6],[-0.121644038467576,0.372786261246687,0.918401460810124,-0.0526487237532504],[-1,0,0,1],[9E+09,9E+09,9E+09,9E+09,9E+09,9E+09]];
	CONST robtarget Target_2320:=[[1346.2,10,-359.6],[-0.120669259343577,0.370470009326083,0.919322472788011,-0.0551098273118455],[-1,0,0,1],[9E+09,9E+09,9E+09,9E+09,9E+09,9E+09]];
	CONST robtarget Target_2330:=[[1346.2,14.9,-359.7],[-0.119702880851243,0.36817161364789,0.920220437906222,-0.0575780242757909],[-1,0,0,1],[9E+09,9E+09,9E+09,9E+09,9E+09,9E+09]];
	CONST robtarget Target_2340:=[[1346.2,19.9,-359.8],[-0.118730850208716,0.365805765459381,0.921128796637897,-0.0600904915091507],[-1,0,0,1],[9E+09,9E+09,9E+09,9E+09,9E+09,9E+09]];
	CONST robtarget Target_2350:=[[1346.2,24.9,-359.9],[-0.117770337947182,0.363418002553263,0.922029378329369,-0.0626045399117393],[-1,0,0,1],[9E+09,9E+09,9E+09,9E+09,9E+09,9E+09]];
	CONST robtarget Target_2360:=[[1346.2,29.8,-360.1],[-0.116849103303759,0.361054468657394,0.922903056228464,-0.0650838422636147],[-1,0,0,1],[9E+09,9E+09,9E+09,9E+09,9E+09,9E+09]];
	CONST robtarget Target_2370:=[[1346.2,34.8,-360.3],[-0.115953593460507,0.358627450987297,0.923783473952652,-0.067566328995428],[-1,0,0,1],[9E+09,9E+09,9E+09,9E+09,9E+09,9E+09]];
	CONST robtarget Target_2380:=[[1346.2,39.8,-360.5],[-0.115039747783415,0.356172521583853,0.924658949304561,-0.0700915028338855],[-1,0,0,1],[9E+09,9E+09,9E+09,9E+09,9E+09,9E+09]];
	CONST robtarget Target_2390:=[[1346.2,44.8,-360.8],[-0.11414938385658,0.353693912795253,0.925524784908103,-0.0726251109297401],[-1,0,0,1],[9E+09,9E+09,9E+09,9E+09,9E+09,9E+09]];
	CONST robtarget Target_2400:=[[1346.2,49.7,-361],[-0.113286516713369,0.351241776432659,0.926365331062547,-0.0751175946417358],[-1,0,0,1],[9E+09,9E+09,9E+09,9E+09,9E+09,9E+09]];
	CONST robtarget Target_2410:=[[1346.2,54.7,-361.3],[-0.112431893149946,0.348716905236613,0.9272131626012,-0.0776617055182264],[-1,0,0,1],[9E+09,9E+09,9E+09,9E+09,9E+09,9E+09]];
	CONST robtarget Target_2420:=[[1346.2,59.7,-361.7],[-0.111608303834052,0.346176237032244,0.928051744458803,-0.0801595848071462],[-1,0,0,1],[9E+09,9E+09,9E+09,9E+09,9E+09,9E+09]];
	CONST robtarget Target_2430:=[[1346.2,64.6,-362.1],[-0.110793593146235,0.343655996914977,0.928865979832894,-0.0826639402109412],[-1,0,0,1],[9E+09,9E+09,9E+09,9E+09,9E+09,9E+09]];
	CONST robtarget Target_2440:=[[1346.2,69.6,-362.5],[-0.109988175498309,0.341061122451655,0.929686704942729,-0.0852205530098301],[-1,0,0,1],[9E+09,9E+09,9E+09,9E+09,9E+09,9E+09]];
	CONST robtarget Target_2450:=[[1346.2,74.6,-362.9],[-0.109196024009588,0.338443041336777,0.93049850140805,-0.0877785565419249],[-1,0,0,1],[9E+09,9E+09,9E+09,9E+09,9E+09,9E+09]];
	CONST robtarget Target_2460:=[[1346.2,79.6,-363.4],[-0.108435328560487,0.3358089775591,0.931301156355231,-0.0902899013295485],[-1,0,0,1],[9E+09,9E+09,9E+09,9E+09,9E+09,9E+09]];
	CONST robtarget Target_2470:=[[1346.2,84.5,-363.8],[-0.107694267553824,0.333194547303151,0.932077470682332,-0.0928166312140292],[-1,0,0,1],[9E+09,9E+09,9E+09,9E+09,9E+09,9E+09]];
	CONST robtarget Target_2480:=[[1346.2,89.5,-364.4],[-0.10695344372535,0.330504885042742,0.93286052701095,-0.0953872055520313],[-1,0,0,1],[9E+09,9E+09,9E+09,9E+09,9E+09,9E+09]];
	CONST robtarget Target_2490:=[[1346.2,94.5,-364.9],[-0.106226744562703,0.327791645339836,0.933634083043202,-0.097958741136734],[-1,0,0,1],[9E+09,9E+09,9E+09,9E+09,9E+09,9E+09]];
	CONST robtarget Target_2500:=[[1346.2,99.5,-365.5],[-0.105542255477612,0.325060026733112,0.934397086557438,-0.100493263266446],[-1,0,0,1],[9E+09,9E+09,9E+09,9E+09,9E+09,9E+09]];
	CONST robtarget Target_2510:=[[1346.2,104.4,-366.1],[-0.10486691842255,0.322351107250489,0.93513458236786,-0.10303400377851],[-1,0,0,1],[9E+09,9E+09,9E+09,9E+09,9E+09,9E+09]];
	CONST robtarget Target_2520:=[[1346.2,109.4,-366.8],[-0.104193781519889,0.319564811629595,0.935877558597188,-0.10561809681534],[-1,0,0,1],[9E+09,9E+09,9E+09,9E+09,9E+09,9E+09]];
	CONST robtarget Target_2530:=[[1346.2,114.4,-367.4],[-0.103545795090149,0.316752112936713,0.936608882026912,-0.108213536018256],[-1,0,0,1],[9E+09,9E+09,9E+09,9E+09,9E+09,9E+09]];
	CONST robtarget Target_2540:=[[1346.2,119.4,-368.1],[-0.102929976384479,0.313922963777386,0.937331090227515,-0.110761997398073],[-1,0,0,1],[9E+09,9E+09,9E+09,9E+09,9E+09,9E+09]];
	CONST robtarget Target_2550:=[[1346.2,124.3,-368.9],[-0.102333534354082,0.311115175405601,0.938025610436359,-0.113327620395202],[-1,0,0,1],[9E+09,9E+09,9E+09,9E+09,9E+09,9E+09]];
	CONST robtarget Target_2560:=[[1346.2,129.3,-369.6],[-0.101741229705465,0.308227713901319,0.938724195658188,-0.115936547503687],[-1,0,0,1],[9E+09,9E+09,9E+09,9E+09,9E+09,9E+09]];
	CONST robtarget Target_2570:=[[1346.2,134.3,-370.4],[-0.101164721884479,0.30531589436779,0.939411916526386,-0.118546002803365],[-1,0,0,1],[9E+09,9E+09,9E+09,9E+09,9E+09,9E+09]];
	CONST robtarget Target_2580:=[[1346.2,139.2,-371.3],[-0.100614451432535,0.302436882539796,0.940074583777804,-0.121113340212912],[-1,0,0,1],[9E+09,9E+09,9E+09,9E+09,9E+09,9E+09]];
	CONST robtarget Target_2590:=[[1346.2,144.2,-372.1],[-0.100079824243535,0.299473728300579,0.940738559926951,-0.123735511085944],[-1,0,0,1],[9E+09,9E+09,9E+09,9E+09,9E+09,9E+09]];
	CONST robtarget Target_2600:=[[1346.2,149.2,-373],[-0.0995877392212445,0.296490765638542,0.941391527592563,-0.126322998162697],[-1,0,0,1],[9E+09,9E+09,9E+09,9E+09,9E+09,9E+09]];
	CONST robtarget Target_2610:=[[1346.2,154.2,-373.9],[-0.0991022967164904,0.293486362708794,0.942034904360776,-0.128898132862591],[-1,0,0,1],[9E+09,9E+09,9E+09,9E+09,9E+09,9E+09]];
	CONST robtarget Target_2620:=[[1346.2,159.1,-374.9],[-0.0986201312562024,0.29049720785679,0.942646751873657,-0.131539131517821],[-1,0,0,1],[9E+09,9E+09,9E+09,9E+09,9E+09,9E+09]];
	CONST robtarget Target_2630:=[[1346.2,164.1,-375.9],[-0.0981717175777088,0.287429251994673,0.943260441132584,-0.134188222881099],[-1,0,0,1],[9E+09,9E+09,9E+09,9E+09,9E+09,9E+09]];
	CONST robtarget Target_2640:=[[1346.2,169.1,-376.9],[-0.0977467849583902,0.284347963494082,0.943866533520709,-0.136776345128341],[-1,0,0,1],[9E+09,9E+09,9E+09,9E+09,9E+09,9E+09]];
	CONST robtarget Target_2650:=[[1346.2,174,-377.9],[-0.0973411284080376,0.281290757965059,0.944442959361686,-0.139383322947305],[-1,0,0,1],[9E+09,9E+09,9E+09,9E+09,9E+09,9E+09]];
	CONST robtarget Target_2660:=[[1341.4,174.3,-376.6],[-0.0970892315469886,0.282881705462646,0.943962262021475,-0.139595378546212],[-1,0,0,1],[9E+09,9E+09,9E+09,9E+09,9E+09,9E+09]];
	CONST robtarget Target_2670:=[[1336.6,174.7,-375.4],[-0.0968578276534226,0.284445199731954,0.943492310384989,-0.139756036778756],[-1,0,0,1],[9E+09,9E+09,9E+09,9E+09,9E+09,9E+09]];
	CONST robtarget Target_2680:=[[1331.9,174.9,-374.1],[-0.0966229425870327,0.286090126554094,0.942991774856666,-0.139939126075453],[-1,0,0,1],[9E+09,9E+09,9E+09,9E+09,9E+09,9E+09]];
	CONST robtarget Target_2690:=[[1327.2,175.2,-372.9],[-0.0963674569829716,0.287694771600429,0.942498051677068,-0.14015154017471],[-1,0,0,1],[9E+09,9E+09,9E+09,9E+09,9E+09,9E+09]];
	CONST robtarget Target_2700:=[[1322.5,175.5,-371.6],[-0.0961248966858667,0.289324553382083,0.94199902432622,-0.140318014580593],[-1,0,0,1],[9E+09,9E+09,9E+09,9E+09,9E+09,9E+09]];
	CONST robtarget Target_2710:=[[1317.8,175.8,-370.4],[-0.0958793438743495,0.290971597327278,0.94149157647326,-0.140485915297344],[-1,0,0,1],[9E+09,9E+09,9E+09,9E+09,9E+09,9E+09]];
	CONST robtarget Target_2720:=[[1313.1,176.1,-369.1],[-0.0956307502487764,0.292636132351492,0.940975532659406,-0.140655254383064],[-1,0,0,1],[9E+09,9E+09,9E+09,9E+09,9E+09,9E+09]];
	CONST robtarget Target_2730:=[[1308.4,176.4,-367.9],[-0.0953627832009456,0.294310263687166,0.940447837135686,-0.140873254719873],[-1,0,0,1],[9E+09,9E+09,9E+09,9E+09,9E+09,9E+09]];
	CONST robtarget Target_2740:=[[1303.6,176.7,-366.6],[-0.095101903278891,0.296050262980581,0.939901541372248,-0.141049503040362],[-1,0,0,1],[9E+09,9E+09,9E+09,9E+09,9E+09,9E+09]];
	CONST robtarget Target_2750:=[[1298.9,177,-365.4],[-0.0948437319418863,0.297769065402197,0.93935842433775,-0.141223230477625],[-1,0,0,1],[9E+09,9E+09,9E+09,9E+09,9E+09,9E+09]];
	CONST robtarget Target_2760:=[[1294.2,177.3,-364.1],[-0.0945657720752437,0.299498165067407,0.938803130092648,-0.141445561264098],[-1,0,0,1],[9E+09,9E+09,9E+09,9E+09,9E+09,9E+09]];
	CONST robtarget Target_2770:=[[1289.5,177.6,-362.9],[-0.0943009704151953,0.301254085156141,0.9382411439109,-0.141622240584786],[-1,0,0,1],[9E+09,9E+09,9E+09,9E+09,9E+09,9E+09]];
	CONST robtarget Target_2780:=[[1284.8,177.9,-361.6],[-0.0940328166867494,0.303028934052148,0.937669415667226,-0.141800428192085],[-1,0,0,1],[9E+09,9E+09,9E+09,9E+09,9E+09,9E+09]];
	CONST robtarget Target_2790:=[[1280.1,178.2,-360.4],[-0.093744445755668,0.304814801264779,0.937084949590598,-0.142027156102845],[-1,0,0,1],[9E+09,9E+09,9E+09,9E+09,9E+09,9E+09]];
	CONST robtarget Target_2800:=[[1275.3,178.5,-359.1],[-0.093462914735115,0.306670511029906,0.936479291540372,-0.142212579436265],[-1,0,0,1],[9E+09,9E+09,9E+09,9E+09,9E+09,9E+09]];
	CONST robtarget Target_2810:=[[1270.6,178.7,-357.9],[-0.0931759327644159,0.30855843130627,0.935858942517041,-0.142400771536465],[-1,0,0,1],[9E+09,9E+09,9E+09,9E+09,9E+09,9E+09]];
	CONST robtarget Target_2820:=[[1265.9,179,-356.6],[-0.0928936110909796,0.310412043924145,0.935245758507429,-0.142585101603138],[-1,0,0,1],[9E+09,9E+09,9E+09,9E+09,9E+09,9E+09]];
	CONST robtarget Target_2830:=[[1261.2,179.3,-355.4],[-0.0925904678703637,0.312277676377353,0.934619019776767,-0.142817876918206],[-1,0,0,1],[9E+09,9E+09,9E+09,9E+09,9E+09,9E+09]];
	CONST robtarget Target_2840:=[[1256.5,179.6,-354.1],[-0.0923098109082863,0.314168238786619,0.933982120911778,-0.143019629299364],[-1,0,0,1],[9E+09,9E+09,9E+09,9E+09,9E+09,9E+09]];
	CONST robtarget Target_2850:=[[1152.7,186.1,-326.6],[-0.0847116064048817,0.361800877254619,0.916546386353804,-0.147874239203031],[-1,0,0,1],[9E+09,9E+09,9E+09,9E+09,9E+09,9E+09]];
	CONST robtarget Target_2860:=[[1148,186.4,-325.4],[-0.0843167371331287,0.364245178298671,0.915577742852347,-0.14809974584311],[-1,0,0,1],[9E+09,9E+09,9E+09,9E+09,9E+09,9E+09]];
	CONST robtarget Target_2870:=[[1143.3,186.7,-324.1],[-0.0839164170034894,0.366716795237724,0.914590588848913,-0.148326942383598],[-1,0,0,1],[9E+09,9E+09,9E+09,9E+09,9E+09,9E+09]];
	CONST robtarget Target_2880:=[[1138.6,187,-322.9],[-0.0834905201851688,0.369207677745856,0.913582291116862,-0.148601551440044],[-1,0,0,1],[9E+09,9E+09,9E+09,9E+09,9E+09,9E+09]];
	CONST robtarget Target_2890:=[[1133.8,187.2,-321.6],[-0.0830604381900551,0.371848073764742,0.912510779106895,-0.148842371853092],[-1,0,0,1],[9E+09,9E+09,9E+09,9E+09,9E+09,9E+09]];
	CONST robtarget Target_2900:=[[1129.1,187.6,-320.4],[-0.082652076021253,0.374348316571166,0.911487931806646,-0.14906952197064],[-1,0,0,1],[9E+09,9E+09,9E+09,9E+09,9E+09,9E+09]];
	CONST robtarget Target_2910:=[[1124.4,187.9,-319.1],[-0.0822084087134797,0.376924329069528,0.910420076965927,-0.149348957644967],[-1,0,0,1],[9E+09,9E+09,9E+09,9E+09,9E+09,9E+09]];
	CONST robtarget Target_2920:=[[1119.7,188.1,-317.9],[-0.081770019911019,0.37959293775452,0.909310655383545,-0.149589429628541],[-1,0,0,1],[9E+09,9E+09,9E+09,9E+09,9E+09,9E+09]];
	CONST robtarget Target_2930:=[[1115,188.4,-316.6],[-0.0813347643139115,0.382235024948745,0.908203199779428,-0.149826532119119],[-1,0,0,1],[9E+09,9E+09,9E+09,9E+09,9E+09,9E+09]];
	CONST robtarget Target_2940:=[[1110.2,188.7,-315.4],[-0.0808833980361246,0.384967105702023,0.907048506924832,-0.150070681796847],[-1,0,0,1],[9E+09,9E+09,9E+09,9E+09,9E+09,9E+09]];
	CONST robtarget Target_2950:=[[1105.5,189,-314.1],[-0.0804148154817876,0.387660313787845,0.905895080873204,-0.150356380026493],[-1,0,0,1],[9E+09,9E+09,9E+09,9E+09,9E+09,9E+09]];
	CONST robtarget Target_2960:=[[1100.8,189.3,-312.9],[-0.0799608049187581,0.390391751395628,0.904721336588572,-0.150598317521762],[-1,0,0,1],[9E+09,9E+09,9E+09,9E+09,9E+09,9E+09]];
	CONST robtarget Target_2970:=[[1096.1,189.6,-311.6],[-0.0795004460623488,0.393153301383706,0.903524708044806,-0.150841846446961],[-1,0,0,1],[9E+09,9E+09,9E+09,9E+09,9E+09,9E+09]];
	CONST robtarget Target_2980:=[[1091.4,189.9,-310.4],[-0.079033646139943,0.395945221351002,0.902304714675516,-0.151086949606733],[-1,0,0,1],[9E+09,9E+09,9E+09,9E+09,9E+09,9E+09]];
	CONST robtarget Target_2990:=[[1086.7,190.2,-309.1],[-0.0785465105296596,0.398755469084056,0.901057401199059,-0.151393795459283],[-1,0,0,1],[9E+09,9E+09,9E+09,9E+09,9E+09,9E+09]];
	CONST robtarget Target_3000:=[[1081.9,190.5,-307.9],[-0.0780554818239111,0.401673398553557,0.899760437713552,-0.151647543261307],[-1,0,0,1],[9E+09,9E+09,9E+09,9E+09,9E+09,9E+09]];
	CONST robtarget Target_3010:=[[1077.2,190.8,-306.6],[-0.077568460848261,0.404558555839991,0.898466882682221,-0.151897233357243],[-1,0,0,1],[9E+09,9E+09,9E+09,9E+09,9E+09,9E+09]];
	CONST robtarget Target_3020:=[[1072.5,191.1,-305.4],[-0.0770746197823937,0.407475053290692,0.897147950633447,-0.152148409802247],[-1,0,0,1],[9E+09,9E+09,9E+09,9E+09,9E+09,9E+09]];
	CONST robtarget Target_3030:=[[1067.8,191.4,-304.1],[-0.0765517619752651,0.4104146743057,0.895801260780301,-0.152445806887078],[-1,0,0,1],[9E+09,9E+09,9E+09,9E+09,9E+09,9E+09]];
	CONST robtarget Target_3040:=[[964,197.8,-276.6],[-0.0633973634082428,0.483924777470896,0.8582888401485,-0.158549206680987],[-1,0,0,1],[9E+09,9E+09,9E+09,9E+09,9E+09,9E+09]];
	CONST robtarget Target_3050:=[[959.3,198.1,-275.4],[-0.0627112764793605,0.487631103520809,0.856188548307434,-0.158821826046096],[-1,0,0,1],[9E+09,9E+09,9E+09,9E+09,9E+09,9E+09]];
	CONST robtarget Target_3060:=[[954.6,198.4,-274.1],[-0.0619901680911656,0.491361119775969,0.854047354893793,-0.159136999567826],[-1,0,0,1],[9E+09,9E+09,9E+09,9E+09,9E+09,9E+09]];
	CONST robtarget Target_3070:=[[949.9,198.7,-272.9],[-0.0612860812394637,0.495131721176396,0.851866898707468,-0.159409478443821],[-1,0,0,1],[9E+09,9E+09,9E+09,9E+09,9E+09,9E+09]];
	CONST robtarget Target_3080:=[[945.2,199,-271.6],[-0.0605730185436125,0.498934034563784,0.849645492886583,-0.159681792938132],[-1,0,0,1],[9E+09,9E+09,9E+09,9E+09,9E+09,9E+09]];
	CONST robtarget Target_3090:=[[940.4,199.3,-270.4],[-0.0598349607407084,0.502852384679912,0.847332351353532,-0.159959816968447],[-1,0,0,1],[9E+09,9E+09,9E+09,9E+09,9E+09,9E+09]];
	CONST robtarget Target_3100:=[[935.7,199.6,-269.1],[-0.0591036477710379,0.506717711523125,0.845026505653726,-0.160231471289439],[-1,0,0,1],[9E+09,9E+09,9E+09,9E+09,9E+09,9E+09]];
	CONST robtarget Target_3110:=[[931,199.9,-267.9],[-0.0583632580352076,0.510613646275031,0.842678075344491,-0.160502634504662],[-1,0,0,1],[9E+09,9E+09,9E+09,9E+09,9E+09,9E+09]];
	CONST robtarget Target_3120:=[[926.3,200.2,-266.6],[-0.0575864775329726,0.514531142755415,0.840285692033365,-0.160814975994649],[-1,0,0,1],[9E+09,9E+09,9E+09,9E+09,9E+09,9E+09]];
	CONST robtarget Target_3130:=[[921.6,200.5,-265.4],[-0.0568276773685659,0.518486941013439,0.837850603090856,-0.16108467954374],[-1,0,0,1],[9E+09,9E+09,9E+09,9E+09,9E+09,9E+09]];
	CONST robtarget Target_3140:=[[916.9,200.8,-264.1],[-0.0560597514291304,0.522471923396913,0.835371432575423,-0.161353534725829],[-1,0,0,1],[9E+09,9E+09,9E+09,9E+09,9E+09,9E+09]];
	CONST robtarget Target_3150:=[[912.1,201.1,-262.9],[-0.055243083445306,0.526561014903931,0.832790323103212,-0.161684807760173],[-1,0,0,1],[9E+09,9E+09,9E+09,9E+09,9E+09,9E+09]];
	CONST robtarget Target_3160:=[[907.4,201.3,-261.6],[-0.0544490363899756,0.530641149913712,0.830196479569303,-0.161953937171013],[-1,0,0,1],[9E+09,9E+09,9E+09,9E+09,9E+09,9E+09]];
	CONST robtarget Target_3170:=[[902.7,201.7,-260.4],[-0.0536606803075758,0.534672785397277,0.827605725709125,-0.162216850906179],[-1,0,0,1],[9E+09,9E+09,9E+09,9E+09,9E+09,9E+09]];
	CONST robtarget Target_3180:=[[898,201.9,-259.1],[-0.0528486753031702,0.538805399750772,0.824921187672144,-0.162483207894506],[-1,0,0,1],[9E+09,9E+09,9E+09,9E+09,9E+09,9E+09]];
	CONST robtarget Target_3190:=[[893.3,202.2,-257.9],[-0.0520348880267262,0.54292686076417,0.822214478425049,-0.162745647428849],[-1,0,0,1],[9E+09,9E+09,9E+09,9E+09,9E+09,9E+09]];
	CONST robtarget Target_3200:=[[888.6,202.5,-256.6],[-0.0511831646230757,0.547064910779842,0.819460739764426,-0.163047119070992],[-1,0,0,1],[9E+09,9E+09,9E+09,9E+09,9E+09,9E+09]];
	CONST robtarget Target_3210:=[[883.8,202.8,-255.4],[-0.0503329330012154,0.551327183738475,0.816599202236212,-0.163311589404054],[-1,0,0,1],[9E+09,9E+09,9E+09,9E+09,9E+09,9E+09]];
	CONST robtarget Target_3220:=[[879.1,203.1,-254.1],[-0.0494918209881874,0.555522322788415,0.81375111029453,-0.16356845366224],[-1,0,0,1],[9E+09,9E+09,9E+09,9E+09,9E+09,9E+09]];
	CONST robtarget Target_3230:=[[775.4,209.6,-226.6],[-0.0287264179271882,0.651799868577542,0.738847368415843,-0.168630633101921],[-1,0,0,1],[9E+09,9E+09,9E+09,9E+09,9E+09,9E+09]];
	CONST robtarget Target_3240:=[[770.6,209.9,-225.3],[-0.0276947373386694,0.656305590777024,0.734847925769366,-0.16880313691109],[-1,0,0,1],[9E+09,9E+09,9E+09,9E+09,9E+09,9E+09]];
	CONST robtarget Target_3250:=[[765.9,210.2,-224.1],[-0.026680029602439,0.660708879169093,0.730891427969873,-0.168966486403946],[-1,0,0,1],[9E+09,9E+09,9E+09,9E+09,9E+09,9E+09]];
	CONST robtarget Target_3260:=[[761.2,210.4,-222.8],[-0.0256597269985173,0.665108223877904,0.726890330808367,-0.169124439149531],[-1,0,0,1],[9E+09,9E+09,9E+09,9E+09,9E+09,9E+09]];
	CONST robtarget Target_3270:=[[756.5,210.7,-221.6],[-0.0246020329108936,0.669481096591472,0.722857684138548,-0.169312048493856],[-1,0,0,1],[9E+09,9E+09,9E+09,9E+09,9E+09,9E+09]];
	CONST robtarget Target_3280:=[[751.8,211,-220.3],[-0.0235754168363021,0.673849886663126,0.718786825460483,-0.169458046458494],[-1,0,0,1],[9E+09,9E+09,9E+09,9E+09,9E+09,9E+09]];
	CONST robtarget Target_3290:=[[747.1,211.3,-219.1],[-0.0225454544995641,0.678204375664533,0.71467964504451,-0.169598149370631],[-1,0,0,1],[9E+09,9E+09,9E+09,9E+09,9E+09,9E+09]];
	CONST robtarget Target_3300:=[[742.3,211.6,-217.8],[-0.0214904506776044,0.682635170651838,0.710448727214428,-0.169735059189927],[-1,0,0,1],[9E+09,9E+09,9E+09,9E+09,9E+09,9E+09]];
	CONST robtarget Target_3310:=[[737.6,211.9,-216.6],[-0.0204547500117696,0.68695586211783,0.706271770435017,-0.169862982990676],[-1,0,0,1],[9E+09,9E+09,9E+09,9E+09,9E+09,9E+09]];
	CONST robtarget Target_3320:=[[732.9,212.2,-215.3],[-0.0193806783205297,0.69124891593368,0.702063223488724,-0.170019280533033],[-1,0,0,1],[9E+09,9E+09,9E+09,9E+09,9E+09,9E+09]];
	CONST robtarget Target_3330:=[[728.2,212.5,-214.1],[-0.0183404329768762,0.695529990609371,0.697822230742038,-0.17013463775303],[-1,0,0,1],[9E+09,9E+09,9E+09,9E+09,9E+09,9E+09]];
	CONST robtarget Target_3340:=[[723.5,212.8,-212.8],[-0.0172985389736161,0.699788967542968,0.693551176525578,-0.170243728209037],[-1,0,0,1],[9E+09,9E+09,9E+09,9E+09,9E+09,9E+09]];
	CONST robtarget Target_3350:=[[718.7,213.1,-211.6],[-0.016233209807903,0.704113910645159,0.689159948336267,-0.17034861121966],[-1,0,0,1],[9E+09,9E+09,9E+09,9E+09,9E+09,9E+09]];
	CONST robtarget Target_3360:=[[714,213.4,-210.3],[-0.0151521984500484,0.708315056353461,0.684833756080143,-0.170478498228622],[-1,0,0,1],[9E+09,9E+09,9E+09,9E+09,9E+09,9E+09]];
	CONST robtarget Target_3370:=[[709.3,213.7,-209.1],[-0.0141072627458021,0.712498254312907,0.680480514140489,-0.170568146539666],[-1,0,0,1],[9E+09,9E+09,9E+09,9E+09,9E+09,9E+09]];
	CONST robtarget Target_3380:=[[704.6,214,-207.8],[-0.0130632722266937,0.716649332376352,0.676103089125091,-0.170668386641371],[-1,0,0,1],[9E+09,9E+09,9E+09,9E+09,9E+09,9E+09]];
	CONST robtarget Target_3390:=[[699.9,214.2,-206.6],[-0.0120203281646521,0.720766616143132,0.671712094407673,-0.170745011613374],[-1,0,0,1],[9E+09,9E+09,9E+09,9E+09,9E+09,9E+09]];
	CONST robtarget Target_3400:=[[695.2,214.6,-205.3],[-0.0109734339531746,0.724870674711254,0.667281168371785,-0.17081548825359],[-1,0,0,1],[9E+09,9E+09,9E+09,9E+09,9E+09,9E+09]];
	CONST robtarget Target_3410:=[[690.4,214.9,-204.1],[-0.00986966433784021,0.729011018321884,0.662747493781276,-0.170913090130001],[-1,0,0,1],[9E+09,9E+09,9E+09,9E+09,9E+09,9E+09]];
	CONST robtarget Target_3420:=[[591.4,4.8,-154.1],[-0.0798329583892878,0.780467197342176,0.610987121559058,-0.105794092068693],[-1,0,0,1],[9E+09,9E+09,9E+09,9E+09,9E+09,9E+09]];
	CONST robtarget Target_3430:=[[591.4,9.6,-154.1],[-0.0779578351486353,0.780856183144148,0.610474569901915,-0.107270670211212],[-1,0,0,1],[9E+09,9E+09,9E+09,9E+09,9E+09,9E+09]];
	CONST robtarget Target_3440:=[[591.4,14.4,-154.2],[-0.0760297502880997,0.78124678844101,0.609953305981917,-0.108765330613513],[-1,0,0,1],[9E+09,9E+09,9E+09,9E+09,9E+09,9E+09]];
	CONST robtarget Target_3450:=[[591.4,19.2,-154.3],[-0.0741448297974858,0.781645170334999,0.609410681540711,-0.110236079077398],[-1,0,0,1],[9E+09,9E+09,9E+09,9E+09,9E+09,9E+09]];
	CONST robtarget Target_3460:=[[591.4,24,-154.4],[-0.0722143009206809,0.782043874937438,0.608857708787523,-0.111735235558803],[-1,0,0,1],[9E+09,9E+09,9E+09,9E+09,9E+09,9E+09]];
	CONST robtarget Target_3470:=[[591.4,28.8,-154.5],[-0.0703193360791187,0.782452363882641,0.608283898159128,-0.113199772385794],[-1,0,0,1],[9E+09,9E+09,9E+09,9E+09,9E+09,9E+09]];
	CONST robtarget Target_3480:=[[591.4,33.6,-154.6],[-0.068378656550929,0.782861391396194,0.60769899721103,-0.114692327460098],[-1,0,0,1],[9E+09,9E+09,9E+09,9E+09,9E+09,9E+09]];
	CONST robtarget Target_3490:=[[591.4,38.4,-154.8],[-0.0664393324379109,0.783274129447367,0.60709693400263,-0.116192796542128],[-1,0,0,1],[9E+09,9E+09,9E+09,9E+09,9E+09,9E+09]];
	CONST robtarget Target_3500:=[[591.4,43.2,-155],[-0.0645289384282897,0.783699196950221,0.606474026715052,-0.117647098242699],[-1,0,0,1],[9E+09,9E+09,9E+09,9E+09,9E+09,9E+09]];
	CONST robtarget Target_3510:=[[591.4,48.1,-155.2],[-0.0625760324051865,0.784137141473964,0.605820411827993,-0.119141983121092],[-1,0,0,1],[9E+09,9E+09,9E+09,9E+09,9E+09,9E+09]];
	CONST robtarget Target_3520:=[[591.4,52.9,-155.4],[-0.0606668659649136,0.784570853997287,0.605161718164253,-0.120612608380934],[-1,0,0,1],[9E+09,9E+09,9E+09,9E+09,9E+09,9E+09]];
	CONST robtarget Target_3530:=[[591.4,57.7,-155.7],[-0.0587051940989133,0.785007458391492,0.604490600771667,-0.122098747062564],[-1,0,0,1],[9E+09,9E+09,9E+09,9E+09,9E+09,9E+09]];
	CONST robtarget Target_3540:=[[591.4,62.5,-156],[-0.0567433477852347,0.785448551764998,0.603800885714858,-0.123593104266963],[-1,0,0,1],[9E+09,9E+09,9E+09,9E+09,9E+09,9E+09]];
	CONST robtarget Target_3550:=[[591.4,67.3,-156.3],[-0.0548110027475357,0.785903705733831,0.603088728165891,-0.125040414470243],[-1,0,0,1],[9E+09,9E+09,9E+09,9E+09,9E+09,9E+09]];
	CONST robtarget Target_3560:=[[591.4,72.1,-156.6],[-0.052837121936533,0.786358349385212,0.602361807327102,-0.126526827081281],[-1,0,0,1],[9E+09,9E+09,9E+09,9E+09,9E+09,9E+09]];
	CONST robtarget Target_3570:=[[591.4,76.9,-156.9],[-0.0509029083013495,0.786823617564496,0.601610989649494,-0.127991038366523],[-1,0,0,1],[9E+09,9E+09,9E+09,9E+09,9E+09,9E+09]];
	CONST robtarget Target_3580:=[[591.4,81.7,-157.3],[-0.04891639017961,0.787292721054174,0.600845318916246,-0.129469150315219],[-1,0,0,1],[9E+09,9E+09,9E+09,9E+09,9E+09,9E+09]];
	CONST robtarget Target_3590:=[[591.4,86.5,-157.7],[-0.0469690862513713,0.787773046546964,0.600055106813583,-0.130925172742933],[-1,0,0,1],[9E+09,9E+09,9E+09,9E+09,9E+09,9E+09]];
	CONST robtarget Target_3600:=[[591.4,91.3,-158.1],[-0.0449696910612702,0.788257682696649,0.599248948941995,-0.132394296506601],[-1,0,0,1],[9E+09,9E+09,9E+09,9E+09,9E+09,9E+09]];
	CONST robtarget Target_3610:=[[591.4,96.1,-158.5],[-0.0429679547082566,0.788748162563807,0.59842161658846,-0.133871803304734],[-1,0,0,1],[9E+09,9E+09,9E+09,9E+09,9E+09,9E+09]];
	CONST robtarget Target_3620:=[[591.4,100.9,-159],[-0.0410043067265913,0.789250700115285,0.597568740998876,-0.135327672626193],[-1,0,0,1],[9E+09,9E+09,9E+09,9E+09,9E+09,9E+09]];
	CONST robtarget Target_3630:=[[591.4,105.7,-159.5],[-0.0389884629030067,0.789758214469715,0.596698248447154,-0.136795697074751],[-1,0,0,1],[9E+09,9E+09,9E+09,9E+09,9E+09,9E+09]];
	CONST robtarget Target_3640:=[[591.4,110.5,-160],[-0.0370101941836127,0.790278453613907,0.595801404484999,-0.138242170461134],[-1,0,0,1],[9E+09,9E+09,9E+09,9E+09,9E+09,9E+09]];
	CONST robtarget Target_3650:=[[591.4,115.3,-160.5],[-0.0349832101977529,0.79080167104292,0.594885658598001,-0.139713797723801],[-1,0,0,1],[9E+09,9E+09,9E+09,9E+09,9E+09,9E+09]];
	CONST robtarget Target_3660:=[[591.4,120.1,-161.1],[-0.0329485449688081,0.791334372979523,0.593946514706166,-0.141180172807449],[-1,0,0,1],[9E+09,9E+09,9E+09,9E+09,9E+09,9E+09]];
	CONST robtarget Target_3670:=[[591.4,124.9,-161.6],[-0.0309473237366203,0.791883429200384,0.592979704952104,-0.142611245090621],[-1,0,0,1],[9E+09,9E+09,9E+09,9E+09,9E+09,9E+09]];
	CONST robtarget Target_3680:=[[591.4,129.7,-162.2],[-0.0288970044197205,0.792436206696833,0.59199209749373,-0.144066574737082],[-1,0,0,1],[9E+09,9E+09,9E+09,9E+09,9E+09,9E+09]];
	CONST robtarget Target_3690:=[[591.4,134.5,-162.8],[-0.0268824469497281,0.793003399287645,0.590975852046503,-0.145500807771452],[-1,0,0,1],[9E+09,9E+09,9E+09,9E+09,9E+09,9E+09]];
	CONST robtarget Target_3700:=[[591.4,139.3,-163.5],[-0.0248181001134522,0.793574732030988,0.589937514922753,-0.146958957112086],[-1,0,0,1],[9E+09,9E+09,9E+09,9E+09,9E+09,9E+09]];
	CONST robtarget Target_3710:=[[591.4,144.1,-164.1],[-0.0227863981041502,0.794164085138318,0.588869330423088,-0.148381594629933],[-1,0,0,1],[9E+09,9E+09,9E+09,9E+09,9E+09,9E+09]];
	CONST robtarget Target_3720:=[[591.4,148.9,-164.8],[-0.0207064803081383,0.794755151650716,0.587777811178003,-0.149842368122943],[-1,0,0,1],[9E+09,9E+09,9E+09,9E+09,9E+09,9E+09]];
	CONST robtarget Target_3730:=[[591.4,153.7,-165.5],[-0.0186155134514777,0.795361089379405,0.586658335789498,-0.151281846924347],[-1,0,0,1],[9E+09,9E+09,9E+09,9E+09,9E+09,9E+09]];
	CONST robtarget Target_3740:=[[591.4,158.5,-166.2],[-0.0165582911969826,0.795983356767578,0.58550734918117,-0.152700565802794],[-1,0,0,1],[9E+09,9E+09,9E+09,9E+09,9E+09,9E+09]];
	CONST robtarget Target_3750:=[[591.4,163.3,-167],[-0.0144500257138868,0.79661118494415,0.584330504449933,-0.154141747583297],[-1,0,0,1],[9E+09,9E+09,9E+09,9E+09,9E+09,9E+09]];
	CONST robtarget Target_3760:=[[591.4,168.1,-167.8],[-0.0123733194837957,0.797259389746827,0.583120492028372,-0.155546964618595],[-1,0,0,1],[9E+09,9E+09,9E+09,9E+09,9E+09,9E+09]];
	CONST robtarget Target_3770:=[[591.4,173,-168.6],[-0.0102403064921214,0.797931716790897,0.581854185872108,-0.156989865421896],[-1,0,0,1],[9E+09,9E+09,9E+09,9E+09,9E+09,9E+09]];
	CONST robtarget Target_3780:=[[591.4,177.8,-169.4],[-0.00814300879571028,0.798607968293856,0.580581266779703,-0.158380545048276],[-1,0,0,1],[9E+09,9E+09,9E+09,9E+09,9E+09,9E+09]];
	CONST robtarget Target_3790:=[[591.4,182.6,-170.2],[-0.00599427406830501,0.799287750768736,0.579279347347488,-0.159808003197952],[-1,0,0,1],[9E+09,9E+09,9E+09,9E+09,9E+09,9E+09]];
	CONST robtarget Target_3800:=[[591.4,187.4,-171.1],[-0.00383447103106639,0.799982326748276,0.577943995973827,-0.161227513905449],[-1,0,0,1],[9E+09,9E+09,9E+09,9E+09,9E+09,9E+09]];
	CONST robtarget Target_3810:=[[591.4,192.2,-172],[-0.00170488325481291,0.800699956846088,0.576571347603175,-0.162610435098181],[-1,0,0,1],[9E+09,9E+09,9E+09,9E+09,9E+09,9E+09]];
	CONST robtarget Target_3820:=[[591.4,197,-172.9],[0.000477917320688526,0.80142199399573,0.575166822061789,-0.164029527629279],[-1,0,0,1],[9E+09,9E+09,9E+09,9E+09,9E+09,9E+09]];
	CONST robtarget Target_3830:=[[591.4,201.8,-173.9],[0.00263137441782939,0.802168157787323,0.573723129592548,-0.165411889147361],[-1,0,0,1],[9E+09,9E+09,9E+09,9E+09,9E+09,9E+09]];
	CONST robtarget Target_3840:=[[591.4,206.6,-174.8],[0.00483819671768203,0.802927124814683,0.572244219860488,-0.166796813295729],[-1,0,0,1],[9E+09,9E+09,9E+09,9E+09,9E+09,9E+09]];
	CONST robtarget Target_3850:=[[591.4,211.4,-175.8],[0.007058994836036,0.803695605988493,0.570727983459168,-0.168205565910661],[-1,0,0,1],[9E+09,9E+09,9E+09,9E+09,9E+09,9E+09]];
	CONST robtarget Target_3860:=[[591.4,216.2,-176.8],[0.00925060229665527,0.804494072471899,0.569168720787369,-0.169560257702086],[-1,0,0,1],[9E+09,9E+09,9E+09,9E+09,9E+09,9E+09]];
	CONST robtarget Target_3870:=[[591.4,221,-177.8],[0.0114983721198495,0.80529879148585,0.567571913689097,-0.17094960269424],[-1,0,0,1],[9E+09,9E+09,9E+09,9E+09,9E+09,9E+09]];
	CONST robtarget Target_3880:=[[596.1,220.7,-179.1],[0.0105444478776632,0.802119716707681,0.572055924579113,-0.171011092744536],[-1,0,0,1],[9E+09,9E+09,9E+09,9E+09,9E+09,9E+09]];
	CONST robtarget Target_3890:=[[600.8,220.4,-180.3],[0.00954125404368884,0.798905975122599,0.576549633518153,-0.171022593462869],[-1,0,0,1],[9E+09,9E+09,9E+09,9E+09,9E+09,9E+09]];
	CONST robtarget Target_3900:=[[605.6,220.1,-181.6],[0.00855378584535725,0.795564255560035,0.581152090482101,-0.171074825007082],[-1,0,0,1],[9E+09,9E+09,9E+09,9E+09,9E+09,9E+09]];
	CONST robtarget Target_3910:=[[610.3,219.8,-182.8],[0.00757988026613238,0.792243418895945,0.5856710699809,-0.171120742222102],[-1,0,0,1],[9E+09,9E+09,9E+09,9E+09,9E+09,9E+09]];
	CONST robtarget Target_3920:=[[615,219.5,-184.1],[0.00659971422524121,0.788876173727834,0.590198796610973,-0.171161347200929],[-1,0,0,1],[9E+09,9E+09,9E+09,9E+09,9E+09,9E+09]];
	CONST robtarget Target_3930:=[[619.7,219.3,-185.3],[0.00561999404124486,0.78548535344611,0.594704125190122,-0.171196316170846],[-1,0,0,1],[9E+09,9E+09,9E+09,9E+09,9E+09,9E+09]];
	CONST robtarget Target_3940:=[[624.4,218.9,-186.6],[0.00458106569260151,0.782012243707725,0.599272432351621,-0.171197010346854],[-1,0,0,1],[9E+09,9E+09,9E+09,9E+09,9E+09,9E+09]];
	CONST robtarget Target_3950:=[[629.1,218.7,-187.8],[0.00358974474052876,0.778529300573558,0.603790299387018,-0.171220665362796],[-1,0,0,1],[9E+09,9E+09,9E+09,9E+09,9E+09,9E+09]];
	CONST robtarget Target_3960:=[[633.9,218.4,-189.1],[0.00256587096633776,0.774905033947616,0.608434701383857,-0.171239069200825],[-1,0,0,1],[9E+09,9E+09,9E+09,9E+09,9E+09,9E+09]];
	CONST robtarget Target_3970:=[[638.6,218.1,-190.3],[0.00155789400513257,0.77131029461782,0.612985339875262,-0.171251205779257],[-1,0,0,1],[9E+09,9E+09,9E+09,9E+09,9E+09,9E+09]];
	CONST robtarget Target_3980:=[[643.3,217.8,-191.6],[0.000505419678604915,0.767680414947257,0.617533589458358,-0.171227307833863],[-1,0,0,1],[9E+09,9E+09,9E+09,9E+09,9E+09,9E+09]];
	CONST robtarget Target_3990:=[[648,217.5,-192.8],[-0.000511535880873687,0.763999243627504,0.62208207604746,-0.171227289671146],[-1,0,0,1],[9E+09,9E+09,9E+09,9E+09,9E+09,9E+09]];
	CONST robtarget Target_4000:=[[652.7,217.2,-194.1],[-0.00153262884980755,0.760275915333536,0.626627071045187,-0.171221194499667],[-1,0,0,1],[9E+09,9E+09,9E+09,9E+09,9E+09,9E+09]];
	CONST robtarget Target_4010:=[[657.4,216.9,-195.3],[-0.00255755580854608,0.756511214628875,0.631166963444428,-0.171208952176486],[-1,0,0,1],[9E+09,9E+09,9E+09,9E+09,9E+09,9E+09]];
	CONST robtarget Target_4020:=[[662.2,216.6,-196.6],[-0.00360764788769451,0.7526256103041,0.63579528491276,-0.171190044318594],[-1,0,0,1],[9E+09,9E+09,9E+09,9E+09,9E+09,9E+09]];
	CONST robtarget Target_4030:=[[666.9,216.3,-197.8],[-0.00467823838086147,0.748788327367839,0.640318160093673,-0.171133891259386],[-1,0,0,1],[9E+09,9E+09,9E+09,9E+09,9E+09,9E+09]];
	CONST robtarget Target_4040:=[[671.6,216,-199.1],[-0.00571266089965787,0.744903909189969,0.644832901937839,-0.171102484369377],[-1,0,0,1],[9E+09,9E+09,9E+09,9E+09,9E+09,9E+09]];
	CONST robtarget Target_4050:=[[676.3,215.7,-200.3],[-0.00674962721138414,0.740981822113494,0.649336002887133,-0.171064716363237],[-1,0,0,1],[9E+09,9E+09,9E+09,9E+09,9E+09,9E+09]];
	CONST robtarget Target_4060:=[[681,215.4,-201.6],[-0.00778880261753513,0.737023119823921,0.65382583781393,-0.171020551998035],[-1,0,0,1],[9E+09,9E+09,9E+09,9E+09,9E+09,9E+09]];
	CONST robtarget Target_4070:=[[685.8,215.1,-202.9],[-0.00885182306103069,0.73294428678642,0.658395001359533,-0.170968827218367],[-1,0,0,1],[9E+09,9E+09,9E+09,9E+09,9E+09,9E+09]];
	CONST robtarget Target_4080:=[[685.8,210.4,-201.8],[-0.0107346225420244,0.732835994506392,0.658916984559389,-0.16930617382089],[-1,0,0,1],[9E+09,9E+09,9E+09,9E+09,9E+09,9E+09]];
	CONST robtarget Target_4090:=[[685.8,205.6,-200.8],[-0.0125762226074915,0.732715789866478,0.659435714163476,-0.167672146735755],[-1,0,0,1],[9E+09,9E+09,9E+09,9E+09,9E+09,9E+09]];
	CONST robtarget Target_4100:=[[685.8,200.8,-199.9],[-0.0144512147493925,0.732607686605116,0.659935499335979,-0.16601890445229],[-1,0,0,1],[9E+09,9E+09,9E+09,9E+09,9E+09,9E+09]];
	CONST robtarget Target_4110:=[[685.8,196,-198.9],[-0.016282557309774,0.732498742412928,0.660420221712942,-0.164394651505338],[-1,0,0,1],[9E+09,9E+09,9E+09,9E+09,9E+09,9E+09]];
	CONST robtarget Target_4120:=[[685.8,191.2,-198],[-0.0181465816081545,0.732404985663715,0.660886618536096,-0.162734495392944],[-1,0,0,1],[9E+09,9E+09,9E+09,9E+09,9E+09,9E+09]];
	CONST robtarget Target_4130:=[[685.8,186.5,-197.1],[-0.0199664997368062,0.732316180721814,0.661327930581443,-0.161120199150018],[-1,0,0,1],[9E+09,9E+09,9E+09,9E+09,9E+09,9E+09]];
	CONST robtarget Target_4140:=[[685.8,181.7,-196.2],[-0.0218201820588689,0.732235039616849,0.661762987697313,-0.159453675172932],[-1,0,0,1],[9E+09,9E+09,9E+09,9E+09,9E+09,9E+09]];
	CONST robtarget Target_4150:=[[685.8,176.9,-195.3],[-0.0236327216680133,0.732148323228141,0.662185106864039,-0.157832859405907],[-1,0,0,1],[9E+09,9E+09,9E+09,9E+09,9E+09,9E+09]];
	CONST robtarget Target_4160:=[[685.8,172.1,-194.5],[-0.0254786508695543,0.732075131676669,0.662590256027763,-0.15617615870394],[-1,0,0,1],[9E+09,9E+09,9E+09,9E+09,9E+09,9E+09]];
	CONST robtarget Target_4170:=[[685.8,167.3,-193.7],[-0.0272817198938289,0.731999530396666,0.66298327537654,-0.15454957725497],[-1,0,0,1],[9E+09,9E+09,9E+09,9E+09,9E+09,9E+09]];
	CONST robtarget Target_4180:=[[685.8,162.6,-192.9],[-0.0290807738548418,0.731934829310175,0.663352315329456,-0.152935999626443],[-1,0,0,1],[9E+09,9E+09,9E+09,9E+09,9E+09,9E+09]];
	CONST robtarget Target_4190:=[[685.8,157.8,-192.1],[-0.0309159204626391,0.731873313330407,0.663715440972814,-0.151286061852978],[-1,0,0,1],[9E+09,9E+09,9E+09,9E+09,9E+09,9E+09]];
	CONST robtarget Target_4200:=[[685.8,153,-191.4],[-0.0327468754827148,0.731816286247317,0.664065082011433,-0.149633325774887],[-1,0,0,1],[9E+09,9E+09,9E+09,9E+09,9E+09,9E+09]];
	CONST robtarget Target_4210:=[[685.8,148.2,-190.7],[-0.0345354927367498,0.731756130198338,0.664404196480068,-0.148011247404572],[-1,0,0,1],[9E+09,9E+09,9E+09,9E+09,9E+09,9E+09]];
	CONST robtarget Target_4220:=[[685.8,143.4,-190],[-0.0363199849090201,0.731700072084409,0.664730600723342,-0.1463867878938],[-1,0,0,1],[9E+09,9E+09,9E+09,9E+09,9E+09,9E+09]];
	CONST robtarget Target_4230:=[[685.8,138.6,-189.3],[-0.0381421845797423,0.731652084921474,0.665041676258664,-0.144741041949451],[-1,0,0,1],[9E+09,9E+09,9E+09,9E+09,9E+09,9E+09]];
	CONST robtarget Target_4240:=[[685.8,133.9,-188.7],[-0.0399589454727848,0.731615674534452,0.665331587380416,-0.143093208385505],[-1,0,0,1],[9E+09,9E+09,9E+09,9E+09,9E+09,9E+09]];
	CONST robtarget Target_4250:=[[685.8,129.1,-188],[-0.0417356050126207,0.731567394271006,0.665621378481879,-0.141476031261997],[-1,0,0,1],[9E+09,9E+09,9E+09,9E+09,9E+09,9E+09]];
	CONST robtarget Target_4260:=[[685.8,124.3,-187.4],[-0.0435085846530386,0.731522357125962,0.665899509006847,-0.139856669454143],[-1,0,0,1],[9E+09,9E+09,9E+09,9E+09,9E+09,9E+09]];
	CONST robtarget Target_4270:=[[685.8,119.5,-186.8],[-0.0453160787115838,0.73148715152165,0.666163137057978,-0.138201573775487],[-1,0,0,1],[9E+09,9E+09,9E+09,9E+09,9E+09,9E+09]];
	CONST robtarget Target_4280:=[[685.8,114.7,-186.3],[-0.0470862410812797,0.731445260227928,0.666418349968379,-0.136591727481413],[-1,0,0,1],[9E+09,9E+09,9E+09,9E+09,9E+09,9E+09]];
	CONST robtarget Target_4290:=[[685.8,110,-185.8],[-0.0488898072835198,0.73142001130423,0.666651333070852,-0.134946485402015],[-1,0,0,1],[9E+09,9E+09,9E+09,9E+09,9E+09,9E+09]];
	CONST robtarget Target_4300:=[[685.8,105.2,-185.2],[-0.0506534174784111,0.731383127475856,0.666884859224499,-0.133332429208026],[-1,0,0,1],[9E+09,9E+09,9E+09,9E+09,9E+09,9E+09]];
	CONST robtarget Target_4310:=[[685.8,100.4,-184.8],[-0.0524569416359899,0.731352644054674,0.667104067491037,-0.131695643228428],[-1,0,0,1],[9E+09,9E+09,9E+09,9E+09,9E+09,9E+09]];
	CONST robtarget Target_4320:=[[685.8,95.6,-184.3],[-0.054214120858505,0.731320186520857,0.6673165746789,-0.130077680812115],[-1,0,0,1],[9E+09,9E+09,9E+09,9E+09,9E+09,9E+09]];
	CONST robtarget Target_4330:=[[685.8,90.8,-183.9],[-0.0560115462076602,0.731293706551634,0.66751495308531,-0.128436789343691],[-1,0,0,1],[9E+09,9E+09,9E+09,9E+09,9E+09,9E+09]];
	CONST robtarget Target_4340:=[[685.8,86.1,-183.4],[-0.0577665836832366,0.731269369491702,0.667699524489086,-0.126828530109849],[-1,0,0,1],[9E+09,9E+09,9E+09,9E+09,9E+09,9E+09]];
	CONST robtarget Target_4350:=[[685.8,81.3,-183],[-0.0595580813182071,0.731246121969508,0.667877945555812,-0.125183840388435],[-1,0,0,1],[9E+09,9E+09,9E+09,9E+09,9E+09,9E+09]];
	CONST robtarget Target_4360:=[[685.8,76.5,-182.7],[-0.0613143717280485,0.73121613510138,0.668049821272029,-0.123583768697206],[-1,0,0,1],[9E+09,9E+09,9E+09,9E+09,9E+09,9E+09]];
	CONST robtarget Target_4370:=[[685.8,71.7,-182.3],[-0.0631000108743183,0.731195641566221,0.668208830495576,-0.121935561793751],[-1,0,0,1],[9E+09,9E+09,9E+09,9E+09,9E+09,9E+09]];
	CONST robtarget Target_4380:=[[685.8,66.9,-182],[-0.0648507783812581,0.731168382720256,0.668361723616571,-0.120331953602846],[-1,0,0,1],[9E+09,9E+09,9E+09,9E+09,9E+09,9E+09]];
	CONST robtarget Target_4390:=[[685.8,62.2,-181.7],[-0.0666358667603735,0.731154172418791,0.668494730207229,-0.118693020438651],[-1,0,0,1],[9E+09,9E+09,9E+09,9E+09,9E+09,9E+09]];
	CONST robtarget Target_4400:=[[685.8,57.4,-181.4],[-0.0683878802063309,0.731127126836983,0.668628704578399,-0.117097726954008],[-1,0,0,1],[9E+09,9E+09,9E+09,9E+09,9E+09,9E+09]];
	CONST robtarget Target_4410:=[[685.8,52.6,-181.1],[-0.070168742508655,0.731108525060423,0.668750207100017,-0.11545489449309],[-1,0,0,1],[9E+09,9E+09,9E+09,9E+09,9E+09,9E+09]];
	CONST robtarget Target_4420:=[[685.8,47.8,-180.9],[-0.0719157425917237,0.731083267284559,0.66886630454598,-0.113856264241447],[-1,0,0,1],[9E+09,9E+09,9E+09,9E+09,9E+09,9E+09]];
	CONST robtarget Target_4430:=[[685.8,43,-180.7],[-0.0736983325234181,0.731064198058668,0.668969354832249,-0.112221639604083],[-1,0,0,1],[9E+09,9E+09,9E+09,9E+09,9E+09,9E+09]];
	CONST robtarget Target_4440:=[[685.8,38.3,-180.5],[-0.0754394523917643,0.731045819187095,0.669062024224519,-0.110620554204403],[-1,0,0,1],[9E+09,9E+09,9E+09,9E+09,9E+09,9E+09]];
	CONST robtarget Target_4450:=[[685.8,33.5,-180.3],[-0.0772170120742314,0.73102754176045,0.669147946907557,-0.108982986669493],[-1,0,0,1],[9E+09,9E+09,9E+09,9E+09,9E+09,9E+09]];
	CONST robtarget Target_4460:=[[685.8,28.7,-180.2],[-0.078961704631492,0.731002764371237,0.669229086083009,-0.107389189510862],[-1,0,0,1],[9E+09,9E+09,9E+09,9E+09,9E+09,9E+09]];
	CONST robtarget Target_4470:=[[685.8,23.9,-180.1],[-0.0807421352151932,0.730983438742031,0.669297304321677,-0.10575934149522],[-1,0,0,1],[9E+09,9E+09,9E+09,9E+09,9E+09,9E+09]];
	CONST robtarget Target_4480:=[[685.8,19.1,-180],[-0.082482290127667,0.730959212820278,0.669361972221373,-0.10416261878605],[-1,0,0,1],[9E+09,9E+09,9E+09,9E+09,9E+09,9E+09]];
	CONST robtarget Target_4490:=[[685.8,14.4,-179.9],[-0.0842193410710339,0.730940266742607,0.669413026608586,-0.102565241922103],[-1,0,0,1],[9E+09,9E+09,9E+09,9E+09,9E+09,9E+09]];
	CONST robtarget Target_4500:=[[685.8,9.6,-179.8],[-0.0860011957234345,0.730919602258051,0.669455884657415,-0.100941309019795],[-1,0,0,1],[9E+09,9E+09,9E+09,9E+09,9E+09,9E+09]];
	CONST robtarget Target_4510:=[[685.8,4.8,-179.8],[-0.0877723447332196,0.730900126075337,0.669491833065371,-0.0993061260036746],[-1,0,0,1],[9E+09,9E+09,9E+09,9E+09,9E+09,9E+09]];
	CONST robtarget Target_4520:=[[690.4,0,-181],[-0.0898851451574911,0.72830728138637,0.672315446183029,-0.0973709678668454],[-1,0,0,1],[9E+09,9E+09,9E+09,9E+09,9E+09,9E+09]];
	CONST robtarget Target_4530:=[[695.2,0,-182.3],[-0.0902736786264436,0.725613803162423,0.675221566566749,-0.0970108635698037],[-1,0,0,1],[9E+09,9E+09,9E+09,9E+09,9E+09,9E+09]];
	CONST robtarget Target_4540:=[[699.9,0,-183.6],[-0.0906531519075061,0.72296217129457,0.678059919309297,-0.0966563539170814],[-1,0,0,1],[9E+09,9E+09,9E+09,9E+09,9E+09,9E+09]];
	CONST robtarget Target_4550:=[[704.6,0,-184.9],[-0.0910316129689519,0.720296750427298,0.680890700935594,-0.0963000007454851],[-1,0,0,1],[9E+09,9E+09,9E+09,9E+09,9E+09,9E+09]];
	CONST robtarget Target_4560:=[[709.3,0,-186.2],[-0.0914090059456191,0.717617874623809,0.68371349359004,-0.0959418487175605],[-1,0,0,1],[9E+09,9E+09,9E+09,9E+09,9E+09,9E+09]];
	CONST robtarget Target_4570:=[[714,0,-187.5],[-0.0917852753980763,0.714925885464751,0.686527882601378,-0.0955819435008976],[-1,0,0,1],[9E+09,9E+09,9E+09,9E+09,9E+09,9E+09]];
	CONST robtarget Target_4580:=[[718.7,0,-188.7],[-0.0921603663591028,0.712221131805988,0.689333456830356,-0.0952203317357456],[-1,0,0,1],[9E+09,9E+09,9E+09,9E+09,9E+09,9E+09]];
	CONST robtarget Target_4590:=[[723.5,0,-190],[-0.0925421650146301,0.709446025389109,0.692189202715765,-0.0948493141657569],[-1,0,0,1],[9E+09,9E+09,9E+09,9E+09,9E+09,9E+09]];
	CONST robtarget Target_4600:=[[728.2,0,-191.3],[-0.092914708248698,0.706716564811144,0.694975720668158,-0.0944843992115567],[-1,0,0,1],[9E+09,9E+09,9E+09,9E+09,9E+09,9E+09]];
	CONST robtarget Target_4610:=[[732.9,0,-192.6],[-0.0932859102524667,0.703975435285204,0.697752206597513,-0.0941179241785443],[-1,0,0,1],[9E+09,9E+09,9E+09,9E+09,9E+09,9E+09]];
	CONST robtarget Target_4620:=[[737.6,0,-193.9],[-0.0936557184145369,0.701223012255294,0.700518266985453,-0.0937499392616681],[-1,0,0,1],[9E+09,9E+09,9E+09,9E+09,9E+09,9E+09]];
	CONST robtarget Target_4630:=[[742.3,0,-195.2],[-0.0940240808191009,0.698459677062998,0.703273513516429,-0.0933804954443521],[-1,0,0,1],[9E+09,9E+09,9E+09,9E+09,9E+09,9E+09]];
	CONST robtarget Target_4640:=[[747.1,0,-196.5],[-0.0943987353020235,0.695626686846901,0.706075823012723,-0.0930017391057177],[-1,0,0,1],[9E+09,9E+09,9E+09,9E+09,9E+09,9E+09]];
	CONST robtarget Target_4650:=[[751.8,0,-197.7],[-0.0947640199710437,0.692842482124379,0.708808048952903,-0.092629505138682],[-1,0,0,1],[9E+09,9E+09,9E+09,9E+09,9E+09,9E+09]];
	CONST robtarget Target_4660:=[[756.5,0,-199],[-0.0951277066760732,0.690048550082335,0.711528322574693,-0.0922559706786529],[-1,0,0,1],[9E+09,9E+09,9E+09,9E+09,9E+09,9E+09]];
	CONST robtarget Target_4670:=[[761.2,0,-200.3],[-0.0954897467097809,0.687245292639746,0.714236279561043,-0.0918811894601467],[-1,0,0,1],[9E+09,9E+09,9E+09,9E+09,9E+09,9E+09]];
	CONST robtarget Target_4680:=[[765.9,0,-201.6],[-0.0958500922589999,0.68443311601584,0.716931562282996,-0.0915052157926022],[-1,0,0,1],[9E+09,9E+09,9E+09,9E+09,9E+09,9E+09]];
	CONST robtarget Target_4690:=[[770.6,0,-202.9],[-0.0962086964404349,0.681612430392518,0.719613820066774,-0.0911281045152467],[-1,0,0,1],[9E+09,9E+09,9E+09,9E+09,9E+09,9E+09]];
	CONST robtarget Target_4700:=[[775.4,0,-204.2],[-0.0965730854348586,0.678723377842014,0.722339346614468,-0.0907418529285191],[-1,0,0,1],[9E+09,9E+09,9E+09,9E+09,9E+09,9E+09]];
	CONST robtarget Target_4710:=[[780.1,4.9,-205.5],[-0.0952732486187487,0.675433915778764,0.725412028727096,-0.0921380599504604],[-1,0,0,1],[9E+09,9E+09,9E+09,9E+09,9E+09,9E+09]];
	CONST robtarget Target_4720:=[[780.1,9.7,-205.5],[-0.0936630902484351,0.674981538894732,0.725818600535032,-0.0938856048272614],[-1,0,0,1],[9E+09,9E+09,9E+09,9E+09,9E+09,9E+09]];
	CONST robtarget Target_4730:=[[780.1,14.6,-205.6],[-0.0920102044366244,0.674513064028716,0.726233604296364,-0.0956608630780421],[-1,0,0,1],[9E+09,9E+09,9E+09,9E+09,9E+09,9E+09]];
	CONST robtarget Target_4740:=[[780.1,19.5,-205.6],[-0.0904024318606843,0.674040590365115,0.726641860850772,-0.0974078483144447],[-1,0,0,1],[9E+09,9E+09,9E+09,9E+09,9E+09,9E+09]];
	CONST robtarget Target_4750:=[[780.1,24.3,-205.8],[-0.0887600400910803,0.673559283615261,0.727049043706982,-0.0991929170026243],[-1,0,0,1],[9E+09,9E+09,9E+09,9E+09,9E+09,9E+09]];
	CONST robtarget Target_4760:=[[780.1,29.2,-205.9],[-0.0871544355703888,0.673070730618972,0.727455195921729,-0.100939753669844],[-1,0,0,1],[9E+09,9E+09,9E+09,9E+09,9E+09,9E+09]];
	CONST robtarget Target_4770:=[[780.1,34.1,-206],[-0.0855584831767584,0.672572467517762,0.727859494761166,-0.10269653246133],[-1,0,0,1],[9E+09,9E+09,9E+09,9E+09,9E+09,9E+09]];
	CONST robtarget Target_4780:=[[780.1,38.9,-206.2],[-0.0839279262167382,0.672064992560099,0.728262506785628,-0.104491483798753],[-1,0,0,1],[9E+09,9E+09,9E+09,9E+09,9E+09,9E+09]];
	CONST robtarget Target_4790:=[[780.1,43.8,-206.4],[-0.0823342777448838,0.671549905840294,0.728665273610882,-0.10624833978797],[-1,0,0,1],[9E+09,9E+09,9E+09,9E+09,9E+09,9E+09]];
	CONST robtarget Target_4800:=[[780.1,48.7,-206.7],[-0.0807070124111121,0.671020367863762,0.7290712143904,-0.108042623102928],[-1,0,0,1],[9E+09,9E+09,9E+09,9E+09,9E+09,9E+09]];
	CONST robtarget Target_4810:=[[780.1,53.5,-206.9],[-0.0790804965520389,0.670487143209706,0.729471752558237,-0.109837279988099],[-1,0,0,1],[9E+09,9E+09,9E+09,9E+09,9E+09,9E+09]];
	CONST robtarget Target_4820:=[[780.1,58.4,-207.2],[-0.0774988954837719,0.669944168816111,0.729871994025955,-0.111604678238241],[-1,0,0,1],[9E+09,9E+09,9E+09,9E+09,9E+09,9E+09]];
	CONST robtarget Target_4830:=[[780.1,63.3,-207.5],[-0.0758838125597801,0.669386050210486,0.730275447335948,-0.113409584221432],[-1,0,0,1],[9E+09,9E+09,9E+09,9E+09,9E+09,9E+09]];
	CONST robtarget Target_4840:=[[780.1,68.1,-207.8],[-0.0743044268335242,0.668830333600852,0.730670223027063,-0.115177524673418],[-1,0,0,1],[9E+09,9E+09,9E+09,9E+09,9E+09,9E+09]];
	CONST robtarget Target_4850:=[[780.1,73,-208.2],[-0.0726927093144144,0.66825372911412,0.731073103013495,-0.116982227657971],[-1,0,0,1],[9E+09,9E+09,9E+09,9E+09,9E+09,9E+09]];
	CONST robtarget Target_4860:=[[780.1,77.9,-208.5],[-0.0711247134818433,0.667671941234459,0.731471984935508,-0.118761059589594],[-1,0,0,1],[9E+09,9E+09,9E+09,9E+09,9E+09,9E+09]];
	CONST robtarget Target_4870:=[[780.1,82.7,-208.9],[-0.0695574926534851,0.667086311805586,0.731865827137734,-0.120540527978694],[-1,0,0,1],[9E+09,9E+09,9E+09,9E+09,9E+09,9E+09]];
	CONST robtarget Target_4880:=[[780.1,87.6,-209.3],[-0.0679582145150368,0.666478713557603,0.732268126041517,-0.122356843037797],[-1,0,0,1],[9E+09,9E+09,9E+09,9E+09,9E+09,9E+09]];
	CONST robtarget Target_4890:=[[780.1,92.5,-209.8],[-0.0663958349758878,0.665867734144869,0.732667785673539,-0.124135690109118],[-1,0,0,1],[9E+09,9E+09,9E+09,9E+09,9E+09,9E+09]];
	CONST robtarget Target_4900:=[[780.1,97.3,-210.3],[-0.0648060627463773,0.665243753910121,0.733064658863416,-0.125964788890968],[-1,0,0,1],[9E+09,9E+09,9E+09,9E+09,9E+09,9E+09]];
	CONST robtarget Target_4910:=[[780.1,102.2,-210.8],[-0.0632193842794307,0.664603304843011,0.733467511396738,-0.127793451978392],[-1,0,0,1],[9E+09,9E+09,9E+09,9E+09,9E+09,9E+09]];
	CONST robtarget Target_4920:=[[780.1,107.1,-211.3],[-0.0616697052210983,0.663959140827434,0.733868432197973,-0.129584840907137],[-1,0,0,1],[9E+09,9E+09,9E+09,9E+09,9E+09,9E+09]];
	CONST robtarget Target_4930:=[[780.1,111.9,-211.8],[-0.0600865013380815,0.663303827631439,0.73426697871006,-0.131414034952253],[-1,0,0,1],[9E+09,9E+09,9E+09,9E+09,9E+09,9E+09]];
	CONST robtarget Target_4940:=[[780.1,116.8,-212.4],[-0.0585473511496776,0.662635655180545,0.734669320300569,-0.133218564644372],[-1,0,0,1],[9E+09,9E+09,9E+09,9E+09,9E+09,9E+09]];
	CONST robtarget Target_4950:=[[780.1,121.7,-213],[-0.0569704354605331,0.661951867549295,0.735075761131224,-0.135047102630122],[-1,0,0,1],[9E+09,9E+09,9E+09,9E+09,9E+09,9E+09]];
	CONST robtarget Target_4960:=[[780.1,126.5,-213.6],[-0.0554404869695827,0.661265382849307,0.735474109068963,-0.136865922489674],[-1,0,0,1],[9E+09,9E+09,9E+09,9E+09,9E+09,9E+09]];
	CONST robtarget Target_4970:=[[780.1,131.4,-214.2],[-0.053874436203336,0.660555964799115,0.735882766190252,-0.138708027584083],[-1,0,0,1],[9E+09,9E+09,9E+09,9E+09,9E+09,9E+09]];
	CONST robtarget Target_4980:=[[780.1,136.3,-214.9],[-0.0523459546611487,0.659842085367383,0.736291003318884,-0.140512924104184],[-1,0,0,1],[9E+09,9E+09,9E+09,9E+09,9E+09,9E+09]];
	CONST robtarget Target_4990:=[[780.1,141.1,-215.6],[-0.0508240535747167,0.659120648257248,0.736694214175996,-0.14233243277198],[-1,0,0,1],[9E+09,9E+09,9E+09,9E+09,9E+09,9E+09]];
	CONST robtarget Target_5000:=[[780.1,146,-216.3],[-0.049272043087392,0.658372098466819,0.73710789605569,-0.144188748877108],[-1,0,0,1],[9E+09,9E+09,9E+09,9E+09,9E+09,9E+09]];
	CONST robtarget Target_5010:=[[780.1,150.9,-217],[-0.0477233167939281,0.657610833647315,0.73752375371748,-0.146045161530081],[-1,0,0,1],[9E+09,9E+09,9E+09,9E+09,9E+09,9E+09]];
	CONST robtarget Target_5020:=[[780.1,155.7,-217.8],[-0.0462153483635271,0.656849010595085,0.737932980259328,-0.14787980085692],[-1,0,0,1],[9E+09,9E+09,9E+09,9E+09,9E+09,9E+09]];
	CONST robtarget Target_5030:=[[780.1,160.6,-218.6],[-0.0446735665735565,0.656061744655232,0.738353755236267,-0.149736407657035],[-1,0,0,1],[9E+09,9E+09,9E+09,9E+09,9E+09,9E+09]];
	CONST robtarget Target_5040:=[[780.1,165.5,-219.4],[-0.0431741622284941,0.655265524072454,0.738775542426874,-0.151571047993333],[-1,0,0,1],[9E+09,9E+09,9E+09,9E+09,9E+09,9E+09]];
	CONST robtarget Target_5050:=[[780.1,170.3,-220.2],[-0.0416424751529547,0.654455959152261,0.739194452157966,-0.153443356624239],[-1,0,0,1],[9E+09,9E+09,9E+09,9E+09,9E+09,9E+09]];
	CONST robtarget Target_5060:=[[780.1,175.2,-221.1],[-0.0401546228730343,0.653628456038539,0.739622371402802,-0.155293900199255],[-1,0,0,1],[9E+09,9E+09,9E+09,9E+09,9E+09,9E+09]];
	CONST robtarget Target_5070:=[[780.1,180.1,-222],[-0.0386364933434536,0.652778237856275,0.74005518049053,-0.157181816354523],[-1,0,0,1],[9E+09,9E+09,9E+09,9E+09,9E+09,9E+09]];
	CONST robtarget Target_5080:=[[780.1,184.9,-222.9],[-0.0371512644850459,0.651933999334024,0.740483060684909,-0.15901786345633],[-1,0,0,1],[9E+09,9E+09,9E+09,9E+09,9E+09,9E+09]];
	CONST robtarget Target_5090:=[[780.1,189.8,-223.8],[-0.0356794135173851,0.651058246767035,0.740922381072643,-0.160885561792642],[-1,0,0,1],[9E+09,9E+09,9E+09,9E+09,9E+09,9E+09]];
	CONST robtarget Target_5100:=[[780.1,194.7,-224.8],[-0.0341746204553322,0.650162231325148,0.741367410884479,-0.162774476971922],[-1,0,0,1],[9E+09,9E+09,9E+09,9E+09,9E+09,9E+09]];
	CONST robtarget Target_5110:=[[780.1,199.5,-225.8],[-0.0326758101233686,0.649255825350651,0.741808275039138,-0.164680441353808],[-1,0,0,1],[9E+09,9E+09,9E+09,9E+09,9E+09,9E+09]];
	CONST robtarget Target_5120:=[[780.1,204.4,-226.8],[-0.0312180242411969,0.64833178533389,0.742261743748568,-0.166549796924472],[-1,0,0,1],[9E+09,9E+09,9E+09,9E+09,9E+09,9E+09]];
	CONST robtarget Target_5130:=[[780.1,209.3,-227.9],[-0.0297315426615164,0.647382132292022,0.742721264864386,-0.168456323354894],[-1,0,0,1],[9E+09,9E+09,9E+09,9E+09,9E+09,9E+09]];
	CONST robtarget Target_5140:=[[784.8,209,-229.1],[-0.0307651390229622,0.642968328984431,0.746552448472756,-0.168239935280534],[-1,0,0,1],[9E+09,9E+09,9E+09,9E+09,9E+09,9E+09]];
	CONST robtarget Target_5150:=[[789.5,208.7,-230.3],[-0.0317593997810374,0.63854274253144,0.750341253269555,-0.168055080636822],[-1,0,0,1],[9E+09,9E+09,9E+09,9E+09,9E+09,9E+09]];
	CONST robtarget Target_5160:=[[794.2,208.4,-231.6],[-0.0327479318751579,0.634115576754324,0.75408637815255,-0.167865251199289],[-1,0,0,1],[9E+09,9E+09,9E+09,9E+09,9E+09,9E+09]];
	CONST robtarget Target_5170:=[[798.9,208.1,-232.8],[-0.0337304773604137,0.629688375941923,0.75778715982875,-0.167670583285617],[-1,0,0,1],[9E+09,9E+09,9E+09,9E+09,9E+09,9E+09]];
	CONST robtarget Target_5180:=[[803.7,207.8,-234.1],[-0.0347604944167214,0.625176161610856,0.761520794777794,-0.16742925103583],[-1,0,0,1],[9E+09,9E+09,9E+09,9E+09,9E+09,9E+09]];
	CONST robtarget Target_5190:=[[808.4,207.5,-235.4],[-0.0357299876826028,0.620753454512114,0.765130252072654,-0.167225040154622],[-1,0,0,1],[9E+09,9E+09,9E+09,9E+09,9E+09,9E+09]];
	CONST robtarget Target_5200:=[[813.1,207.2,-236.6],[-0.0366892387091784,0.616339415627857,0.768694156957296,-0.166999753191925],[-1,0,0,1],[9E+09,9E+09,9E+09,9E+09,9E+09,9E+09]];
	CONST robtarget Target_5210:=[[817.8,206.9,-237.8],[-0.0376450070876776,0.611927170340272,0.772211188986617,-0.166786903696278],[-1,0,0,1],[9E+09,9E+09,9E+09,9E+09,9E+09,9E+09]];
	CONST robtarget Target_5220:=[[822.5,206.6,-239.1],[-0.0385936457931231,0.607522308703406,0.775681395048548,-0.166569950193959],[-1,0,0,1],[9E+09,9E+09,9E+09,9E+09,9E+09,9E+09]];
	CONST robtarget Target_5230:=[[827.3,206.3,-240.3],[-0.0395868816896496,0.603040074957237,0.779177750824128,-0.166305680643543],[-1,0,0,1],[9E+09,9E+09,9E+09,9E+09,9E+09,9E+09]];
	CONST robtarget Target_5240:=[[832,206,-241.6],[-0.0405203170220552,0.598654293350079,0.782552449639827,-0.166080716895896],[-1,0,0,1],[9E+09,9E+09,9E+09,9E+09,9E+09,9E+09]];
	CONST robtarget Target_5250:=[[836.7,205.7,-242.8],[-0.0414460623868268,0.594280009004696,0.785879488395744,-0.165852116443685],[-1,0,0,1],[9E+09,9E+09,9E+09,9E+09,9E+09,9E+09]];
	CONST robtarget Target_5260:=[[841.4,205.5,-244.1],[-0.042369168495389,0.589893666567888,0.789177268759606,-0.165618701169982],[-1,0,0,1],[9E+09,9E+09,9E+09,9E+09,9E+09,9E+09]];
	CONST robtarget Target_5270:=[[846.1,205.2,-245.3],[-0.0432792420588702,0.585545172332437,0.792409080300039,-0.165383215058337],[-1,0,0,1],[9E+09,9E+09,9E+09,9E+09,9E+09,9E+09]];
	CONST robtarget Target_5280:=[[850.8,204.9,-246.6],[-0.0442117627725604,0.58122061137896,0.795592994627718,-0.165105141773693],[-1,0,0,1],[9E+09,9E+09,9E+09,9E+09,9E+09,9E+09]];
	CONST robtarget Target_5290:=[[855.5,204.6,-247.9],[-0.0451051805643158,0.576903849032486,0.798728715624983,-0.164863308512928],[-1,0,0,1],[9E+09,9E+09,9E+09,9E+09,9E+09,9E+09]];
	CONST robtarget Target_5300:=[[860.2,204.3,-249.1],[-0.0459901904631258,0.572604680792359,0.801816370328713,-0.16461862041924],[-1,0,0,1],[9E+09,9E+09,9E+09,9E+09,9E+09,9E+09]];
	CONST robtarget Target_5310:=[[865,204,-250.3],[-0.0468856267688857,0.568231430194026,0.804921520355919,-0.164365829204422],[-1,0,0,1],[9E+09,9E+09,9E+09,9E+09,9E+09,9E+09]];
	CONST robtarget Target_5320:=[[869.7,203.7,-251.6],[-0.0477830710999151,0.563979721183965,0.807912615766751,-0.164075767541839],[-1,0,0,1],[9E+09,9E+09,9E+09,9E+09,9E+09,9E+09]];
	CONST robtarget Target_5330:=[[874.5,203.4,-252.9],[-0.0486604304958268,0.559648139841036,0.810919157619479,-0.16381770930563],[-1,0,0,1],[9E+09,9E+09,9E+09,9E+09,9E+09,9E+09]];
	CONST robtarget Target_5340:=[[874.5,198.6,-251.8],[-0.0497288829466965,0.561614453537066,0.809896265744502,-0.16181558179683],[-1,0,0,1],[9E+09,9E+09,9E+09,9E+09,9E+09,9E+09]];
	CONST robtarget Target_5350:=[[874.5,193.7,-250.8],[-0.0508300547284465,0.563585326175979,0.808866135353661,-0.15976063574439],[-1,0,0,1],[9E+09,9E+09,9E+09,9E+09,9E+09,9E+09]];
	CONST robtarget Target_5360:=[[874.5,188.9,-249.8],[-0.051931076153332,0.565471372220381,0.807868525659351,-0.157777488184286],[-1,0,0,1],[9E+09,9E+09,9E+09,9E+09,9E+09,9E+09]];
	CONST robtarget Target_5370:=[[874.5,184,-248.9],[-0.0530643647709649,0.567362551934756,0.806863337796103,-0.155741651378387],[-1,0,0,1],[9E+09,9E+09,9E+09,9E+09,9E+09,9E+09]];
	CONST robtarget Target_5380:=[[874.5,179.2,-248],[-0.0542212915705561,0.569184908836263,0.805889858811547,-0.153720937279803],[-1,0,0,1],[9E+09,9E+09,9E+09,9E+09,9E+09,9E+09]];
	CONST robtarget Target_5390:=[[874.5,174.3,-247.1],[-0.0553551772270953,0.570992543887626,0.804908159170705,-0.151743779046526],[-1,0,0,1],[9E+09,9E+09,9E+09,9E+09,9E+09,9E+09]];
	CONST robtarget Target_5400:=[[874.5,169.5,-246.2],[-0.0565061582642222,0.572738455609367,0.803957595697304,-0.149766150598279],[-1,0,0,1],[9E+09,9E+09,9E+09,9E+09,9E+09,9E+09]];
	CONST robtarget Target_5410:=[[874.5,164.6,-245.3],[-0.0576937442447817,0.574486654555024,0.802998110444125,-0.147751650536835],[-1,0,0,1],[9E+09,9E+09,9E+09,9E+09,9E+09,9E+09]];
	CONST robtarget Target_5420:=[[874.5,159.8,-244.5],[-0.0588726953198289,0.576164563797454,0.8020680702951,-0.145791672543263],[-1,0,0,1],[9E+09,9E+09,9E+09,9E+09,9E+09,9E+09]];
	CONST robtarget Target_5430:=[[874.5,155,-243.7],[-0.0600926947560273,0.577819751108963,0.801147227102332,-0.143792641576606],[-1,0,0,1],[9E+09,9E+09,9E+09,9E+09,9E+09,9E+09]];
	CONST robtarget Target_5440:=[[874.5,150.1,-242.9],[-0.0612881023354137,0.579462021422162,0.800218564873319,-0.14183716957678],[-1,0,0,1],[9E+09,9E+09,9E+09,9E+09,9E+09,9E+09]];
	CONST robtarget Target_5450:=[[874.5,145.3,-242.2],[-0.0625345519472289,0.581054314575751,0.79931592179258,-0.139854819346857],[-1,0,0,1],[9E+09,9E+09,9E+09,9E+09,9E+09,9E+09]];
	CONST robtarget Target_5460:=[[874.5,140.4,-241.4],[-0.0637805022625367,0.582645101885721,0.79840521250172,-0.137861704000058],[-1,0,0,1],[9E+09,9E+09,9E+09,9E+09,9E+09,9E+09]];
	CONST robtarget Target_5470:=[[874.5,135.6,-240.7],[-0.0650154852096765,0.584172927949053,0.797521257970306,-0.135922110121354],[-1,0,0,1],[9E+09,9E+09,9E+09,9E+09,9E+09,9E+09]];
	CONST robtarget Target_5480:=[[874.5,130.8,-240.1],[-0.0662966460814902,0.585678484858534,0.796643616641608,-0.133956765996858],[-1,0,0,1],[9E+09,9E+09,9E+09,9E+09,9E+09,9E+09]];
	CONST robtarget Target_5490:=[[874.5,125.9,-239.4],[-0.06754561054412,0.587175490569763,0.795759308551243,-0.132021424868949],[-1,0,0,1],[9E+09,9E+09,9E+09,9E+09,9E+09,9E+09]];
	CONST robtarget Target_5500:=[[874.5,121.1,-238.8],[-0.0688443221916565,0.588628431763588,0.794897416222129,-0.130058165083529],[-1,0,0,1],[9E+09,9E+09,9E+09,9E+09,9E+09,9E+09]];
	CONST robtarget Target_5510:=[[874.5,116.2,-238.2],[-0.0701168251174381,0.590070517418566,0.794028344192764,-0.128138221961024],[-1,0,0,1],[9E+09,9E+09,9E+09,9E+09,9E+09,9E+09]];
	CONST robtarget Target_5520:=[[874.5,111.4,-237.6],[-0.0714318790139884,0.591473245402668,0.793181072008647,-0.126177151816723],[-1,0,0,1],[9E+09,9E+09,9E+09,9E+09,9E+09,9E+09]];
	CONST robtarget Target_5530:=[[874.5,106.6,-237.1],[-0.0727234602264129,0.592844681903098,0.792342426654749,-0.12425763716881],[-1,0,0,1],[9E+09,9E+09,9E+09,9E+09,9E+09,9E+09]];
	CONST robtarget Target_5540:=[[874.5,101.7,-236.5],[-0.0740575087603239,0.594217826791605,0.791492358416587,-0.122313148465022],[-1,0,0,1],[9E+09,9E+09,9E+09,9E+09,9E+09,9E+09]];
	CONST robtarget Target_5550:=[[874.5,96.9,-236],[-0.0753708930809926,0.595540146201833,0.790666213919857,-0.120408059961581],[-1,0,0,1],[9E+09,9E+09,9E+09,9E+09,9E+09,9E+09]];
	CONST robtarget Target_5560:=[[874.5,92,-235.5],[-0.0767195522825399,0.596866743684801,0.789829162157336,-0.118465586507262],[-1,0,0,1],[9E+09,9E+09,9E+09,9E+09,9E+09,9E+09]];
